   VAR
      sFB_Displacement010 { ExternalAccessible := 'False'; ExternalVisible := 'False'; ExternalWritable := 'False'; S7_SetPoint := 'False'} : "FB_Displacement";   // Displacement calculation for 010 conveyor
      sFB_Displacement020 { ExternalAccessible := 'False'; ExternalVisible := 'False'; ExternalWritable := 'False'; S7_SetPoint := 'False'} : "FB_Displacement";   // Displacement calculation for 020 conveyor
      sFB_Displacement030 { ExternalAccessible := 'False'; ExternalVisible := 'False'; ExternalWritable := 'False'; S7_SetPoint := 'False'} : "FB_Displacement";   // Displacement calculation for 030 conveyor
      sFB_Displacement040 { ExternalAccessible := 'False'; ExternalVisible := 'False'; ExternalWritable := 'False'; S7_SetPoint := 'False'} : "FB_Displacement";   // Displacement calculation for 040 conveyor
      sFB_Displacement050 { ExternalAccessible := 'False'; ExternalVisible := 'False'; ExternalWritable := 'False'; S7_SetPoint := 'False'} : "FB_Displacement";   // Displacement calculation for 050 conveyor
      sFB_Displacement060 { ExternalAccessible := 'False'; ExternalVisible := 'False'; ExternalWritable := 'False'; S7_SetPoint := 'False'} : "FB_Displacement";   // Displacement calculation for 060 conveyor
      sFB_Displacement070 { ExternalAccessible := 'False'; ExternalVisible := 'False'; ExternalWritable := 'False'; S7_SetPoint := 'False'} : "FB_Displacement";   // Displacement calculation for 070 conveyor
      sFB_Displacement080 { ExternalAccessible := 'False'; ExternalVisible := 'False'; ExternalWritable := 'False'; S7_SetPoint := 'False'} : "FB_Displacement";   // Displacement calculation for 080 conveyor
      sFB_Displacement090 { ExternalAccessible := 'False'; ExternalVisible := 'False'; ExternalWritable := 'False'; S7_SetPoint := 'False'} : "FB_Displacement";   // Displacement calculation for 090 conveyor
      sFB_Displacement100 { ExternalAccessible := 'False'; ExternalVisible := 'False'; ExternalWritable := 'False'; S7_SetPoint := 'False'} : "FB_Displacement";   // Displacement calculation for 100 conveyor
      sFB_Displacement110 { ExternalAccessible := 'False'; ExternalVisible := 'False'; ExternalWritable := 'False'; S7_SetPoint := 'False'} : "FB_Displacement";   // Displacement calculation for 110 conveyor
      sFB_Displacement120 { ExternalAccessible := 'False'; ExternalVisible := 'False'; ExternalWritable := 'False'; S7_SetPoint := 'False'} : "FB_Displacement";   // Displacement calculation for 120 conveyor
      sFB_Displacement121 { ExternalAccessible := 'False'; ExternalVisible := 'False'; ExternalWritable := 'False'; S7_SetPoint := 'False'} : "FB_Displacement";   // Displacement calculation for 121 conveyor
      sFB_Displacement210 { ExternalAccessible := 'False'; ExternalVisible := 'False'; ExternalWritable := 'False'; S7_SetPoint := 'False'} : "FB_Displacement";   // Displacement calculation for 210 conveyor
      sFB_Displacement220 { ExternalAccessible := 'False'; ExternalVisible := 'False'; ExternalWritable := 'False'; S7_SetPoint := 'False'} : "FB_Displacement";   // Displacement calculation for 220 conveyor
      sFB_Displacement221 { ExternalAccessible := 'False'; ExternalVisible := 'False'; ExternalWritable := 'False'; S7_SetPoint := 'False'} : "FB_Displacement";   // Displacement calculation for 221 conveyor
      sFB_Displacement230 { ExternalAccessible := 'False'; ExternalVisible := 'False'; ExternalWritable := 'False'; S7_SetPoint := 'False'} : "FB_Displacement";   // Displacement calculation for 230 conveyor
      sFB_Displacement240 { ExternalAccessible := 'False'; ExternalVisible := 'False'; ExternalWritable := 'False'; S7_SetPoint := 'False'} : "FB_Displacement";   // Displacement calculation for 240 conveyor
      sFB_Displacement250 { ExternalAccessible := 'False'; ExternalVisible := 'False'; ExternalWritable := 'False'; S7_SetPoint := 'False'} : "FB_Displacement";   // Displacement calculation for 250 conveyor
      sFB_Displacement260 { ExternalAccessible := 'False'; ExternalVisible := 'False'; ExternalWritable := 'False'; S7_SetPoint := 'False'} : "FB_Displacement";   // Displacement calculation for 260 conveyor
      sFB_Displacement270 { ExternalAccessible := 'False'; ExternalVisible := 'False'; ExternalWritable := 'False'; S7_SetPoint := 'False'} : "FB_Displacement";   // Displacement calculation for 270 conveyor
      sFB_Displacement280 { ExternalAccessible := 'False'; ExternalVisible := 'False'; ExternalWritable := 'False'; S7_SetPoint := 'False'} : "FB_Displacement";   // Displacement calculation for 280 conveyor
      sFB_Displacement290 { ExternalAccessible := 'False'; ExternalVisible := 'False'; ExternalWritable := 'False'; S7_SetPoint := 'False'} : "FB_Displacement";   // Displacement calculation for 290 conveyor
      sFB_Displacement291 { ExternalAccessible := 'False'; ExternalVisible := 'False'; ExternalWritable := 'False'; S7_SetPoint := 'False'} : "FB_Displacement";   // Displacement calculation for 291 conveyor
      sFB_Displacement300 { ExternalAccessible := 'False'; ExternalVisible := 'False'; ExternalWritable := 'False'; S7_SetPoint := 'False'} : "FB_Displacement";   // Displacement calculation for 300 conveyor
      sFB_Displacement410 { ExternalAccessible := 'False'; ExternalVisible := 'False'; ExternalWritable := 'False'; S7_SetPoint := 'False'} : "FB_Displacement";   // Displacement calculation for 410 conveyor
      sFB_Displacement420 { ExternalAccessible := 'False'; ExternalVisible := 'False'; ExternalWritable := 'False'; S7_SetPoint := 'False'} : "FB_Displacement";   // Displacement calculation for 420 conveyor
      sFB_Displacement421 { ExternalAccessible := 'False'; ExternalVisible := 'False'; ExternalWritable := 'False'; S7_SetPoint := 'False'} : "FB_Displacement";   // Displacement calculation for 421 conveyor
      sFB_Displacement430 { ExternalAccessible := 'False'; ExternalVisible := 'False'; ExternalWritable := 'False'; S7_SetPoint := 'False'} : "FB_Displacement";   // Displacement calculation for 430 conveyor
      sFB_Displacement440 { ExternalAccessible := 'False'; ExternalVisible := 'False'; ExternalWritable := 'False'; S7_SetPoint := 'False'} : "FB_Displacement";   // Displacement calculation for 440 conveyor
      sFB_Displacement450 { ExternalAccessible := 'False'; ExternalVisible := 'False'; ExternalWritable := 'False'; S7_SetPoint := 'False'} : "FB_Displacement";   // Displacement calculation for 450 conveyor
      sFB_Displacement460 { ExternalAccessible := 'False'; ExternalVisible := 'False'; ExternalWritable := 'False'; S7_SetPoint := 'False'} : "FB_Displacement";   // Displacement calculation for 460 conveyor
      sFB_Displacement470 { ExternalAccessible := 'False'; ExternalVisible := 'False'; ExternalWritable := 'False'; S7_SetPoint := 'False'} : "FB_Displacement";   // Displacement calculation for 470 conveyor
      sFB_Displacement480 { ExternalAccessible := 'False'; ExternalVisible := 'False'; ExternalWritable := 'False'; S7_SetPoint := 'False'} : "FB_Displacement";   // Displacement calculation for 480 conveyor
      sFB_Displacement490 { ExternalAccessible := 'False'; ExternalVisible := 'False'; ExternalWritable := 'False'; S7_SetPoint := 'False'} : "FB_Displacement";   // Displacement calculation for 490 conveyor
      sFB_Displacement491 { ExternalAccessible := 'False'; ExternalVisible := 'False'; ExternalWritable := 'False'; S7_SetPoint := 'False'} : "FB_Displacement";   // Displacement calculation for 491 conveyor
      sFB_Displacement500 { ExternalAccessible := 'False'; ExternalVisible := 'False'; ExternalWritable := 'False'; S7_SetPoint := 'False'} : "FB_Displacement";   // Displacement calculation for 500 conveyor
      sFB_Displacement610 { ExternalAccessible := 'False'; ExternalVisible := 'False'; ExternalWritable := 'False'; S7_SetPoint := 'False'} : "FB_Displacement";   // Displacement calculation for 610 conveyor
      sFB_Displacement611 { ExternalAccessible := 'False'; ExternalVisible := 'False'; ExternalWritable := 'False'; S7_SetPoint := 'False'} : "FB_Displacement";   // Displacement calculation for 611 conveyor
      sFB_Displacement620 { ExternalAccessible := 'False'; ExternalVisible := 'False'; ExternalWritable := 'False'; S7_SetPoint := 'False'} : "FB_Displacement";   // Displacement calculation for 620 conveyor
      sFB_Displacement630 { ExternalAccessible := 'False'; ExternalVisible := 'False'; ExternalWritable := 'False'; S7_SetPoint := 'False'} : "FB_Displacement";   // Displacement calculation for 630 conveyor
      sFB_Displacement640 { ExternalAccessible := 'False'; ExternalVisible := 'False'; ExternalWritable := 'False'; S7_SetPoint := 'False'} : "FB_Displacement";   // Displacement calculation for 640 conveyor
      sUDT_Interface010 { ExternalAccessible := 'False'; ExternalVisible := 'False'; ExternalWritable := 'False'; S7_SetPoint := 'False'} : "UDT_ConveyorInterface";   // Interface structure for 010 conveyor
      sUDT_Interface020 { ExternalAccessible := 'False'; ExternalVisible := 'False'; ExternalWritable := 'False'; S7_SetPoint := 'False'} : "UDT_ConveyorInterface";   // Interface structure for 020 conveyor
      sUDT_Interface030 { ExternalAccessible := 'False'; ExternalVisible := 'False'; ExternalWritable := 'False'; S7_SetPoint := 'False'} : "UDT_ConveyorInterface";   // Interface structure for 030 conveyor
      sUDT_Interface040 { ExternalAccessible := 'False'; ExternalVisible := 'False'; ExternalWritable := 'False'; S7_SetPoint := 'False'} : "UDT_ConveyorInterface";   // Interface structure for 040 conveyor
      sUDT_Interface050 { ExternalAccessible := 'False'; ExternalVisible := 'False'; ExternalWritable := 'False'; S7_SetPoint := 'False'} : "UDT_ConveyorInterface";   // Interface structure for 050 conveyor
      sUDT_Interface060 { ExternalAccessible := 'False'; ExternalVisible := 'False'; ExternalWritable := 'False'; S7_SetPoint := 'False'} : "UDT_ConveyorInterface";   // Interface structure for 060 conveyor
      sUDT_Interface070 { ExternalAccessible := 'False'; ExternalVisible := 'False'; ExternalWritable := 'False'; S7_SetPoint := 'False'} : "UDT_ConveyorInterface";   // Interface structure for 070 conveyor
      sUDT_Interface080 { ExternalAccessible := 'False'; ExternalVisible := 'False'; ExternalWritable := 'False'; S7_SetPoint := 'False'} : "UDT_ConveyorInterface";   // Interface structure for 080 conveyor
      sUDT_Interface090 { ExternalAccessible := 'False'; ExternalVisible := 'False'; ExternalWritable := 'False'; S7_SetPoint := 'False'} : "UDT_ConveyorInterface";   // Interface structure for 090 conveyor
      sUDT_Interface100 { ExternalAccessible := 'False'; ExternalVisible := 'False'; ExternalWritable := 'False'; S7_SetPoint := 'False'} : "UDT_ConveyorInterface";   // Interface structure for 100 conveyor
      sUDT_Interface110 { ExternalAccessible := 'False'; ExternalVisible := 'False'; ExternalWritable := 'False'; S7_SetPoint := 'False'} : "UDT_ConveyorInterface";   // Interface structure for 110 conveyor
      sUDT_Interface120 { ExternalAccessible := 'False'; ExternalVisible := 'False'; ExternalWritable := 'False'; S7_SetPoint := 'False'} : "UDT_ConveyorInterface";   // Interface structure for 120 conveyor
      sUDT_Interface121 { ExternalAccessible := 'False'; ExternalVisible := 'False'; ExternalWritable := 'False'; S7_SetPoint := 'False'} : "UDT_ConveyorInterface";   // Interface structure for 121 conveyor
      sUDT_Interface210 { ExternalAccessible := 'False'; ExternalVisible := 'False'; ExternalWritable := 'False'; S7_SetPoint := 'False'} : "UDT_ConveyorInterface";   // Interface structure for 210 conveyor
      sUDT_Interface220 { ExternalAccessible := 'False'; ExternalVisible := 'False'; ExternalWritable := 'False'; S7_SetPoint := 'False'} : "UDT_ConveyorInterface";   // Interface structure for 220 conveyor
      sUDT_Interface221 { ExternalAccessible := 'False'; ExternalVisible := 'False'; ExternalWritable := 'False'; S7_SetPoint := 'False'} : "UDT_ConveyorInterface";   // Interface structure for 221 conveyor
      sUDT_Interface230 { ExternalAccessible := 'False'; ExternalVisible := 'False'; ExternalWritable := 'False'; S7_SetPoint := 'False'} : "UDT_ConveyorInterface";   // Interface structure for 230 conveyor
      sUDT_Interface240 { ExternalAccessible := 'False'; ExternalVisible := 'False'; ExternalWritable := 'False'; S7_SetPoint := 'False'} : "UDT_ConveyorInterface";   // Interface structure for 240 conveyor
      sUDT_Interface250 { ExternalAccessible := 'False'; ExternalVisible := 'False'; ExternalWritable := 'False'; S7_SetPoint := 'False'} : "UDT_ConveyorInterface";   // Interface structure for 250 conveyor
      sUDT_Interface260 { ExternalAccessible := 'False'; ExternalVisible := 'False'; ExternalWritable := 'False'; S7_SetPoint := 'False'} : "UDT_ConveyorInterface";   // Interface structure for 260 conveyor
      sUDT_Interface270 { ExternalAccessible := 'False'; ExternalVisible := 'False'; ExternalWritable := 'False'; S7_SetPoint := 'False'} : "UDT_ConveyorInterface";   // Interface structure for 270 conveyor
      sUDT_Interface280 { ExternalAccessible := 'False'; ExternalVisible := 'False'; ExternalWritable := 'False'; S7_SetPoint := 'False'} : "UDT_ConveyorInterface";   // Interface structure for 280 conveyor
      sUDT_Interface290 { ExternalAccessible := 'False'; ExternalVisible := 'False'; ExternalWritable := 'False'; S7_SetPoint := 'False'} : "UDT_ConveyorInterface";   // Interface structure for 290 conveyor
      sUDT_Interface291 { ExternalAccessible := 'False'; ExternalVisible := 'False'; ExternalWritable := 'False'; S7_SetPoint := 'False'} : "UDT_ConveyorInterface";   // Interface structure for 291 conveyor
      sUDT_Interface300 { ExternalAccessible := 'False'; ExternalVisible := 'False'; ExternalWritable := 'False'; S7_SetPoint := 'False'} : "UDT_ConveyorInterface";   // Interface structure for 300 conveyor
      sUDT_Interface410 { ExternalAccessible := 'False'; ExternalVisible := 'False'; ExternalWritable := 'False'; S7_SetPoint := 'False'} : "UDT_ConveyorInterface";   // Interface structure for 410 conveyor
      sUDT_Interface420 { ExternalAccessible := 'False'; ExternalVisible := 'False'; ExternalWritable := 'False'; S7_SetPoint := 'False'} : "UDT_ConveyorInterface";   // Interface structure for 420 conveyor
      sUDT_Interface421 { ExternalAccessible := 'False'; ExternalVisible := 'False'; ExternalWritable := 'False'; S7_SetPoint := 'False'} : "UDT_ConveyorInterface";   // Interface structure for 421 conveyor
      sUDT_Interface430 { ExternalAccessible := 'False'; ExternalVisible := 'False'; ExternalWritable := 'False'; S7_SetPoint := 'False'} : "UDT_ConveyorInterface";   // Interface structure for 430 conveyor
      sUDT_Interface440 { ExternalAccessible := 'False'; ExternalVisible := 'False'; ExternalWritable := 'False'; S7_SetPoint := 'False'} : "UDT_ConveyorInterface";   // Interface structure for 440 conveyor
      sUDT_Interface450 { ExternalAccessible := 'False'; ExternalVisible := 'False'; ExternalWritable := 'False'; S7_SetPoint := 'False'} : "UDT_ConveyorInterface";   // Interface structure for 450 conveyor
      sUDT_Interface460 { ExternalAccessible := 'False'; ExternalVisible := 'False'; ExternalWritable := 'False'; S7_SetPoint := 'False'} : "UDT_ConveyorInterface";   // Interface structure for 460 conveyor
      sUDT_Interface470 { ExternalAccessible := 'False'; ExternalVisible := 'False'; ExternalWritable := 'False'; S7_SetPoint := 'False'} : "UDT_ConveyorInterface";   // Interface structure for 470 conveyor
      sUDT_Interface480 { ExternalAccessible := 'False'; ExternalVisible := 'False'; ExternalWritable := 'False'; S7_SetPoint := 'False'} : "UDT_ConveyorInterface";   // Interface structure for 480 conveyor
      sUDT_Interface490 { ExternalAccessible := 'False'; ExternalVisible := 'False'; ExternalWritable := 'False'; S7_SetPoint := 'False'} : "UDT_ConveyorInterface";   // Interface structure for 490 conveyor
      sUDT_Interface491 { ExternalAccessible := 'False'; ExternalVisible := 'False'; ExternalWritable := 'False'; S7_SetPoint := 'False'} : "UDT_ConveyorInterface";   // Interface structure for 491 conveyor
      sUDT_Interface500 { ExternalAccessible := 'False'; ExternalVisible := 'False'; ExternalWritable := 'False'; S7_SetPoint := 'False'} : "UDT_ConveyorInterface";   // Interface structure for 500 conveyor
      sUDT_Interface610 { ExternalAccessible := 'False'; ExternalVisible := 'False'; ExternalWritable := 'False'; S7_SetPoint := 'False'} : "UDT_ConveyorInterface";   // Interface structure for 610 conveyor
      sUDT_Interface611 { ExternalAccessible := 'False'; ExternalVisible := 'False'; ExternalWritable := 'False'; S7_SetPoint := 'False'} : "UDT_ConveyorInterface";   // Interface structure for 611 conveyor
      sUDT_Interface620 { ExternalAccessible := 'False'; ExternalVisible := 'False'; ExternalWritable := 'False'; S7_SetPoint := 'False'} : "UDT_ConveyorInterface";   // Interface structure for 620 conveyor
      sUDT_Interface630 { ExternalAccessible := 'False'; ExternalVisible := 'False'; ExternalWritable := 'False'; S7_SetPoint := 'False'} : "UDT_ConveyorInterface";   // Interface structure for 630 conveyor
      sUDT_Interface640 { ExternalAccessible := 'False'; ExternalVisible := 'False'; ExternalWritable := 'False'; S7_SetPoint := 'False'} : "UDT_ConveyorInterface";   // Interface structure for 640 conveyor
      sUDT_Handshake010 { ExternalAccessible := 'False'; ExternalVisible := 'False'; ExternalWritable := 'False'; S7_SetPoint := 'False'} : "UDT_ConveyorHandshake";   // Handshake structure for 010 conveyor
      sUDT_Handshake020 { ExternalAccessible := 'False'; ExternalVisible := 'False'; ExternalWritable := 'False'; S7_SetPoint := 'False'} : "UDT_ConveyorHandshake";   // Handshake structure for 020 conveyor
      sUDT_Handshake030 { ExternalAccessible := 'False'; ExternalVisible := 'False'; ExternalWritable := 'False'; S7_SetPoint := 'False'} : "UDT_ConveyorHandshake";   // Handshake structure for 030 conveyor
      sUDT_Handshake040 { ExternalAccessible := 'False'; ExternalVisible := 'False'; ExternalWritable := 'False'; S7_SetPoint := 'False'} : "UDT_ConveyorHandshake";   // Handshake structure for 040 conveyor
      sUDT_Handshake050 { ExternalAccessible := 'False'; ExternalVisible := 'False'; ExternalWritable := 'False'; S7_SetPoint := 'False'} : "UDT_ConveyorHandshake";   // Handshake structure for 050 conveyor
      sUDT_Handshake060 { ExternalAccessible := 'False'; ExternalVisible := 'False'; ExternalWritable := 'False'; S7_SetPoint := 'False'} : "UDT_ConveyorHandshake";   // Handshake structure for 060 conveyor
      sUDT_Handshake070 { ExternalAccessible := 'False'; ExternalVisible := 'False'; ExternalWritable := 'False'; S7_SetPoint := 'False'} : "UDT_ConveyorHandshake";   // Handshake structure for 070 conveyor
      sUDT_Handshake080 { ExternalAccessible := 'False'; ExternalVisible := 'False'; ExternalWritable := 'False'; S7_SetPoint := 'False'} : "UDT_ConveyorHandshake";   // Handshake structure for 080 conveyor
      sUDT_Handshake090 { ExternalAccessible := 'False'; ExternalVisible := 'False'; ExternalWritable := 'False'; S7_SetPoint := 'False'} : "UDT_ConveyorHandshake";   // Handshake structure for 090 conveyor
      sUDT_Handshake100 { ExternalAccessible := 'False'; ExternalVisible := 'False'; ExternalWritable := 'False'; S7_SetPoint := 'False'} : "UDT_ConveyorHandshake";   // Handshake structure for 100 conveyor
      sUDT_Handshake110 { ExternalAccessible := 'False'; ExternalVisible := 'False'; ExternalWritable := 'False'; S7_SetPoint := 'False'} : "UDT_ConveyorHandshake";   // Handshake structure for 110 conveyor
      sUDT_Handshake120 { ExternalAccessible := 'False'; ExternalVisible := 'False'; ExternalWritable := 'False'; S7_SetPoint := 'False'} : "UDT_ConveyorHandshake";   // Handshake structure for 120 conveyor
      sUDT_Handshake121 { ExternalAccessible := 'False'; ExternalVisible := 'False'; ExternalWritable := 'False'; S7_SetPoint := 'False'} : "UDT_ConveyorHandshake";   // Handshake structure for 121 conveyor
      sUDT_HandshakeUp121 { ExternalAccessible := 'False'; ExternalVisible := 'False'; ExternalWritable := 'False'; S7_SetPoint := 'False'} : "UDT_ConveyorHandshake";   // HandshakeUp structure for 121 conveyor
      sUDT_Handshake210 { ExternalAccessible := 'False'; ExternalVisible := 'False'; ExternalWritable := 'False'; S7_SetPoint := 'False'} : "UDT_ConveyorHandshake";   // Handshake structure for 210 conveyor
      sUDT_Handshake220 { ExternalAccessible := 'False'; ExternalVisible := 'False'; ExternalWritable := 'False'; S7_SetPoint := 'False'} : "UDT_ConveyorHandshake";   // Handshake structure for 220 conveyor
      sUDT_Handshake221 { ExternalAccessible := 'False'; ExternalVisible := 'False'; ExternalWritable := 'False'; S7_SetPoint := 'False'} : "UDT_ConveyorHandshake";   // Handshake structure for 221 conveyor
      sUDT_Handshake230 { ExternalAccessible := 'False'; ExternalVisible := 'False'; ExternalWritable := 'False'; S7_SetPoint := 'False'} : "UDT_ConveyorHandshake";   // Handshake structure for 230 conveyor
      sUDT_Handshake240 { ExternalAccessible := 'False'; ExternalVisible := 'False'; ExternalWritable := 'False'; S7_SetPoint := 'False'} : "UDT_ConveyorHandshake";   // Handshake structure for 240 conveyor
      sUDT_Handshake250 { ExternalAccessible := 'False'; ExternalVisible := 'False'; ExternalWritable := 'False'; S7_SetPoint := 'False'} : "UDT_ConveyorHandshake";   // Handshake structure for 250 conveyor
      sUDT_Handshake260 { ExternalAccessible := 'False'; ExternalVisible := 'False'; ExternalWritable := 'False'; S7_SetPoint := 'False'} : "UDT_ConveyorHandshake";   // Handshake structure for 260 conveyor
      sUDT_Handshake270 { ExternalAccessible := 'False'; ExternalVisible := 'False'; ExternalWritable := 'False'; S7_SetPoint := 'False'} : "UDT_ConveyorHandshake";   // Handshake structure for 270 conveyor
      sUDT_Handshake280 { ExternalAccessible := 'False'; ExternalVisible := 'False'; ExternalWritable := 'False'; S7_SetPoint := 'False'} : "UDT_ConveyorHandshake";   // Handshake structure for 280 conveyor
      sUDT_Handshake290 { ExternalAccessible := 'False'; ExternalVisible := 'False'; ExternalWritable := 'False'; S7_SetPoint := 'False'} : "UDT_ConveyorHandshake";   // Handshake structure for 290 conveyor
      sUDT_Handshake291 { ExternalAccessible := 'False'; ExternalVisible := 'False'; ExternalWritable := 'False'; S7_SetPoint := 'False'} : "UDT_ConveyorHandshake";   // Handshake structure for 291 conveyor
      sUDT_HandshakeUp291 { ExternalAccessible := 'False'; ExternalVisible := 'False'; ExternalWritable := 'False'; S7_SetPoint := 'False'} : "UDT_ConveyorHandshake";   // HandshakeUp structure for 291 conveyor
      sUDT_Handshake300 { ExternalAccessible := 'False'; ExternalVisible := 'False'; ExternalWritable := 'False'; S7_SetPoint := 'False'} : "UDT_ConveyorHandshake";   // Handshake structure for 300 conveyor
      sUDT_Handshake410 { ExternalAccessible := 'False'; ExternalVisible := 'False'; ExternalWritable := 'False'; S7_SetPoint := 'False'} : "UDT_ConveyorHandshake";   // Handshake structure for 410 conveyor
      sUDT_Handshake420 { ExternalAccessible := 'False'; ExternalVisible := 'False'; ExternalWritable := 'False'; S7_SetPoint := 'False'} : "UDT_ConveyorHandshake";   // Handshake structure for 420 conveyor
      sUDT_Handshake421 { ExternalAccessible := 'False'; ExternalVisible := 'False'; ExternalWritable := 'False'; S7_SetPoint := 'False'} : "UDT_ConveyorHandshake";   // Handshake structure for 421 conveyor
      sUDT_Handshake430 { ExternalAccessible := 'False'; ExternalVisible := 'False'; ExternalWritable := 'False'; S7_SetPoint := 'False'} : "UDT_ConveyorHandshake";   // Handshake structure for 430 conveyor
      sUDT_Handshake440 { ExternalAccessible := 'False'; ExternalVisible := 'False'; ExternalWritable := 'False'; S7_SetPoint := 'False'} : "UDT_ConveyorHandshake";   // Handshake structure for 440 conveyor
      sUDT_Handshake450 { ExternalAccessible := 'False'; ExternalVisible := 'False'; ExternalWritable := 'False'; S7_SetPoint := 'False'} : "UDT_ConveyorHandshake";   // Handshake structure for 450 conveyor
      sUDT_Handshake460 { ExternalAccessible := 'False'; ExternalVisible := 'False'; ExternalWritable := 'False'; S7_SetPoint := 'False'} : "UDT_ConveyorHandshake";   // Handshake structure for 460 conveyor
      sUDT_Handshake470 { ExternalAccessible := 'False'; ExternalVisible := 'False'; ExternalWritable := 'False'; S7_SetPoint := 'False'} : "UDT_ConveyorHandshake";   // Handshake structure for 470 conveyor
      sUDT_Handshake480 { ExternalAccessible := 'False'; ExternalVisible := 'False'; ExternalWritable := 'False'; S7_SetPoint := 'False'} : "UDT_ConveyorHandshake";   // Handshake structure for 480 conveyor
      sUDT_Handshake490 { ExternalAccessible := 'False'; ExternalVisible := 'False'; ExternalWritable := 'False'; S7_SetPoint := 'False'} : "UDT_ConveyorHandshake";   // Handshake structure for 490 conveyor
      sUDT_Handshake491 { ExternalAccessible := 'False'; ExternalVisible := 'False'; ExternalWritable := 'False'; S7_SetPoint := 'False'} : "UDT_ConveyorHandshake";   // Handshake structure for 491 conveyor
      sUDT_Handshake500 { ExternalAccessible := 'False'; ExternalVisible := 'False'; ExternalWritable := 'False'; S7_SetPoint := 'False'} : "UDT_ConveyorHandshake";   // Handshake structure for 500 conveyor
      sUDT_Handshake610 { ExternalAccessible := 'False'; ExternalVisible := 'False'; ExternalWritable := 'False'; S7_SetPoint := 'False'} : "UDT_ConveyorHandshake";   // Handshake structure for 610 conveyor
      sUDT_Handshake611 { ExternalAccessible := 'False'; ExternalVisible := 'False'; ExternalWritable := 'False'; S7_SetPoint := 'False'} : "UDT_ConveyorHandshake";   // Handshake structure for 611 conveyor
      sUDT_Handshake620 { ExternalAccessible := 'False'; ExternalVisible := 'False'; ExternalWritable := 'False'; S7_SetPoint := 'False'} : "UDT_ConveyorHandshake";   // Handshake structure for 620 conveyor
      sUDT_Handshake630 { ExternalAccessible := 'False'; ExternalVisible := 'False'; ExternalWritable := 'False'; S7_SetPoint := 'False'} : "UDT_ConveyorHandshake";   // Handshake structure for 630 conveyor
      sUDT_Handshake640 { ExternalAccessible := 'False'; ExternalVisible := 'False'; ExternalWritable := 'False'; S7_SetPoint := 'False'} : "UDT_ConveyorHandshake";   // Handshake structure for 640 conveyor
      sFB_PEC010 { ExternalAccessible := 'False'; ExternalVisible := 'False'; ExternalWritable := 'False'; S7_SetPoint := 'False'} : "FB_PEC";   // Photoeye handling for 010 conveyor
      sFB_PEC020 { ExternalAccessible := 'False'; ExternalVisible := 'False'; ExternalWritable := 'False'; S7_SetPoint := 'False'} : "FB_PEC";   // Photoeye handling for 020 conveyor
      sFB_PEC040 { ExternalAccessible := 'False'; ExternalVisible := 'False'; ExternalWritable := 'False'; S7_SetPoint := 'False'} : "FB_PEC";   // Photoeye handling for 040 conveyor
      sFB_PEC050 { ExternalAccessible := 'False'; ExternalVisible := 'False'; ExternalWritable := 'False'; S7_SetPoint := 'False'} : "FB_PEC";   // Photoeye handling for 050 conveyor
      sFB_PEC060 { ExternalAccessible := 'False'; ExternalVisible := 'False'; ExternalWritable := 'False'; S7_SetPoint := 'False'} : "FB_PEC";   // Photoeye handling for 060 conveyor
      sFB_PEC070 { ExternalAccessible := 'False'; ExternalVisible := 'False'; ExternalWritable := 'False'; S7_SetPoint := 'False'} : "FB_PEC";   // Photoeye handling for 070 conveyor
      sFB_PEC080 { ExternalAccessible := 'False'; ExternalVisible := 'False'; ExternalWritable := 'False'; S7_SetPoint := 'False'} : "FB_PEC";   // Photoeye handling for 080 conveyor
      sFB_PEC100 { ExternalAccessible := 'False'; ExternalVisible := 'False'; ExternalWritable := 'False'; S7_SetPoint := 'False'} : "FB_PEC";   // Photoeye handling for 100 conveyor
      sFB_PEC110 { ExternalAccessible := 'False'; ExternalVisible := 'False'; ExternalWritable := 'False'; S7_SetPoint := 'False'} : "FB_PEC";   // Photoeye handling for 110 conveyor
      sFB_PEC120 { ExternalAccessible := 'False'; ExternalVisible := 'False'; ExternalWritable := 'False'; S7_SetPoint := 'False'} : "FB_PEC";   // Photoeye handling for 120 conveyor
      sFB_PEC210 { ExternalAccessible := 'False'; ExternalVisible := 'False'; ExternalWritable := 'False'; S7_SetPoint := 'False'} : "FB_PEC";   // Photoeye handling for 210 conveyor
      sFB_PEC220 { ExternalAccessible := 'False'; ExternalVisible := 'False'; ExternalWritable := 'False'; S7_SetPoint := 'False'} : "FB_PEC";   // Photoeye handling for 220 conveyor
      sFB_PEC240 { ExternalAccessible := 'False'; ExternalVisible := 'False'; ExternalWritable := 'False'; S7_SetPoint := 'False'} : "FB_PEC";   // Photoeye handling for 240 conveyor
      sFB_PEC250 { ExternalAccessible := 'False'; ExternalVisible := 'False'; ExternalWritable := 'False'; S7_SetPoint := 'False'} : "FB_PEC";   // Photoeye handling for 250 conveyor
      sFB_PEC260 { ExternalAccessible := 'False'; ExternalVisible := 'False'; ExternalWritable := 'False'; S7_SetPoint := 'False'} : "FB_PEC";   // Photoeye handling for 260 conveyor
      sFB_PEC280 { ExternalAccessible := 'False'; ExternalVisible := 'False'; ExternalWritable := 'False'; S7_SetPoint := 'False'} : "FB_PEC";   // Photoeye handling for 280 conveyor
      sFB_PEC290 { ExternalAccessible := 'False'; ExternalVisible := 'False'; ExternalWritable := 'False'; S7_SetPoint := 'False'} : "FB_PEC";   // Photoeye handling for 290 conveyor
      sFB_PEC300 { ExternalAccessible := 'False'; ExternalVisible := 'False'; ExternalWritable := 'False'; S7_SetPoint := 'False'} : "FB_PEC";   // Photoeye handling for 3000 conveyor
      sFB_PEC410 { ExternalAccessible := 'False'; ExternalVisible := 'False'; ExternalWritable := 'False'; S7_SetPoint := 'False'} : "FB_PEC";   // Photoeye handling for 410 conveyor
      sFB_PEC420 { ExternalAccessible := 'False'; ExternalVisible := 'False'; ExternalWritable := 'False'; S7_SetPoint := 'False'} : "FB_PEC";   // Photoeye handling for 420 conveyor
      sFB_PEC440 { ExternalAccessible := 'False'; ExternalVisible := 'False'; ExternalWritable := 'False'; S7_SetPoint := 'False'} : "FB_PEC";   // Photoeye handling for 440 conveyor
      sFB_PEC450 { ExternalAccessible := 'False'; ExternalVisible := 'False'; ExternalWritable := 'False'; S7_SetPoint := 'False'} : "FB_PEC";   // Photoeye handling for 450 conveyor
      sFB_PEC460 { ExternalAccessible := 'False'; ExternalVisible := 'False'; ExternalWritable := 'False'; S7_SetPoint := 'False'} : "FB_PEC";   // Photoeye handling for 460 conveyor
      sFB_PEC480 { ExternalAccessible := 'False'; ExternalVisible := 'False'; ExternalWritable := 'False'; S7_SetPoint := 'False'} : "FB_PEC";   // Photoeye handling for 480 conveyor
      sFB_PEC490 { ExternalAccessible := 'False'; ExternalVisible := 'False'; ExternalWritable := 'False'; S7_SetPoint := 'False'} : "FB_PEC";   // Photoeye handling for 490 conveyor
      sFB_PEC500 { ExternalAccessible := 'False'; ExternalVisible := 'False'; ExternalWritable := 'False'; S7_SetPoint := 'False'} : "FB_PEC";   // Photoeye handling for 500 conveyor
      sFB_PEC610 { ExternalAccessible := 'False'; ExternalVisible := 'False'; ExternalWritable := 'False'; S7_SetPoint := 'False'} : "FB_PEC";   // Photoeye handling for 610 conveyor
      sFB_PEC640 { ExternalAccessible := 'False'; ExternalVisible := 'False'; ExternalWritable := 'False'; S7_SetPoint := 'False'} : "FB_PEC";   // Photoeye handling for 640 conveyor
      sFB_Conveyor010 { ExternalAccessible := 'False'; ExternalVisible := 'False'; ExternalWritable := 'False'; S7_SetPoint := 'False'} : "FB_Conveyor";   // Function block to control the 010 conveyor
      sFB_Conveyor020 { ExternalAccessible := 'False'; ExternalVisible := 'False'; ExternalWritable := 'False'; S7_SetPoint := 'False'} : "FB_Conveyor";   // Function block to control the 020 conveyor
      sFB_Conveyor030 { ExternalAccessible := 'False'; ExternalVisible := 'False'; ExternalWritable := 'False'; S7_SetPoint := 'False'} : "FB_Conveyor";   // Function block to control the 030 conveyor
      sFB_Conveyor040 { ExternalAccessible := 'False'; ExternalVisible := 'False'; ExternalWritable := 'False'; S7_SetPoint := 'False'} : "FB_Conveyor";   // Function block to control the 040 conveyor
      sFB_Conveyor050 { ExternalAccessible := 'False'; ExternalVisible := 'False'; ExternalWritable := 'False'; S7_SetPoint := 'False'} : "FB_Conveyor";   // Function block to control the 050 conveyor
      sFB_Conveyor060 { ExternalAccessible := 'False'; ExternalVisible := 'False'; ExternalWritable := 'False'; S7_SetPoint := 'False'} : "FB_Conveyor";   // Function block to control the 060 conveyor
      sFB_Conveyor070 { ExternalAccessible := 'False'; ExternalVisible := 'False'; ExternalWritable := 'False'; S7_SetPoint := 'False'} : "FB_Conveyor";   // Function block to control the 070 conveyor
      sFB_Conveyor080 { ExternalAccessible := 'False'; ExternalVisible := 'False'; ExternalWritable := 'False'; S7_SetPoint := 'False'} : "FB_Conveyor";   // Function block to control the 080 conveyor
      sFB_Conveyor090 { ExternalAccessible := 'False'; ExternalVisible := 'False'; ExternalWritable := 'False'; S7_SetPoint := 'False'} : "FB_Conveyor";   // Function block to control the 090 conveyor
      sFB_Conveyor100 { ExternalAccessible := 'False'; ExternalVisible := 'False'; ExternalWritable := 'False'; S7_SetPoint := 'False'} : "FB_Conveyor";   // Function block to control the 100 conveyor
      sFB_Conveyor110 { ExternalAccessible := 'False'; ExternalVisible := 'False'; ExternalWritable := 'False'; S7_SetPoint := 'False'} : "FB_Conveyor";   // Function block to control the 110 conveyor
      sFB_Conveyor210 { ExternalAccessible := 'False'; ExternalVisible := 'False'; ExternalWritable := 'False'; S7_SetPoint := 'False'} : "FB_Conveyor";   // Function block to control the 210 conveyor
      sFB_Conveyor230 { ExternalAccessible := 'False'; ExternalVisible := 'False'; ExternalWritable := 'False'; S7_SetPoint := 'False'} : "FB_Conveyor";   // Function block to control the 230 conveyor
      sFB_Conveyor240 { ExternalAccessible := 'False'; ExternalVisible := 'False'; ExternalWritable := 'False'; S7_SetPoint := 'False'} : "FB_Conveyor";   // Function block to control the 240 conveyor
      sFB_Conveyor250 { ExternalAccessible := 'False'; ExternalVisible := 'False'; ExternalWritable := 'False'; S7_SetPoint := 'False'} : "FB_Conveyor";   // Function block to control the 250 conveyor
      sFB_Conveyor260 { ExternalAccessible := 'False'; ExternalVisible := 'False'; ExternalWritable := 'False'; S7_SetPoint := 'False'} : "FB_Conveyor";   // Function block to control the 260 conveyor
      sFB_Conveyor270 { ExternalAccessible := 'False'; ExternalVisible := 'False'; ExternalWritable := 'False'; S7_SetPoint := 'False'} : "FB_Conveyor";   // Function block to control the 270 conveyor
      sFB_Conveyor280 { ExternalAccessible := 'False'; ExternalVisible := 'False'; ExternalWritable := 'False'; S7_SetPoint := 'False'} : "FB_Conveyor";   // Function block to control the 280 conveyor
      sFB_Conveyor300 { ExternalAccessible := 'False'; ExternalVisible := 'False'; ExternalWritable := 'False'; S7_SetPoint := 'False'} : "FB_Conveyor";   // Function block to control the 300 conveyor
      sFB_Conveyor410 { ExternalAccessible := 'False'; ExternalVisible := 'False'; ExternalWritable := 'False'; S7_SetPoint := 'False'} : "FB_Conveyor";   // Function block to control the 410 conveyor
      sFB_Conveyor430 { ExternalAccessible := 'False'; ExternalVisible := 'False'; ExternalWritable := 'False'; S7_SetPoint := 'False'} : "FB_Conveyor";   // Function block to control the 430 conveyor
      sFB_Conveyor440 { ExternalAccessible := 'False'; ExternalVisible := 'False'; ExternalWritable := 'False'; S7_SetPoint := 'False'} : "FB_Conveyor";   // Function block to control the 440 conveyor
      sFB_Conveyor450 { ExternalAccessible := 'False'; ExternalVisible := 'False'; ExternalWritable := 'False'; S7_SetPoint := 'False'} : "FB_Conveyor";   // Function block to control the 450 conveyor
      sFB_Conveyor460 { ExternalAccessible := 'False'; ExternalVisible := 'False'; ExternalWritable := 'False'; S7_SetPoint := 'False'} : "FB_Conveyor";   // Function block to control the 460 conveyor
      sFB_Conveyor470 { ExternalAccessible := 'False'; ExternalVisible := 'False'; ExternalWritable := 'False'; S7_SetPoint := 'False'} : "FB_Conveyor";   // Function block to control the 470 conveyor
      sFB_Conveyor480 { ExternalAccessible := 'False'; ExternalVisible := 'False'; ExternalWritable := 'False'; S7_SetPoint := 'False'} : "FB_Conveyor";   // Function block to control the 480 conveyor
      sFB_Conveyor500 { ExternalAccessible := 'False'; ExternalVisible := 'False'; ExternalWritable := 'False'; S7_SetPoint := 'False'} : "FB_Conveyor";   // Function block to control the 500 conveyor
      sFB_Conveyor620 { ExternalAccessible := 'False'; ExternalVisible := 'False'; ExternalWritable := 'False'; S7_SetPoint := 'False'} : "FB_Conveyor";   // Function block to control the 620 conveyor
      sFB_Conveyor630 { ExternalAccessible := 'False'; ExternalVisible := 'False'; ExternalWritable := 'False'; S7_SetPoint := 'False'} : "FB_Conveyor";   // Function block to control the 630 conveyor
      sFB_Conveyor640 { ExternalAccessible := 'False'; ExternalVisible := 'False'; ExternalWritable := 'False'; S7_SetPoint := 'False'} : "FB_Conveyor";   // Function block to control the 640 conveyor
      sFB_MCOConveyLinxAixController010 { ExternalAccessible := 'False'; ExternalVisible := 'False'; ExternalWritable := 'False'; S7_SetPoint := 'False'} : "FB_MCOConveyLinxAixController";   // Function to interface with ConveyLinx Aix Controller for 010
      sFB_MCOConveyLinxAixController020 { ExternalAccessible := 'False'; ExternalVisible := 'False'; ExternalWritable := 'False'; S7_SetPoint := 'False'} : "FB_MCOConveyLinxAixController";   // Function to interface with ConveyLinx Aix Controller for 020
      sFB_MCOConveyLinxAixController030 { ExternalAccessible := 'False'; ExternalVisible := 'False'; ExternalWritable := 'False'; S7_SetPoint := 'False'} : "FB_MCOConveyLinxAixController";   // Function to interface with ConveyLinx Aix Controller for 030
      sFB_MCOConveyLinxAixController040 { ExternalAccessible := 'False'; ExternalVisible := 'False'; ExternalWritable := 'False'; S7_SetPoint := 'False'} : "FB_MCOConveyLinxAixController";   // Function to interface with ConveyLinx Aix Controller for 040
      sFB_MCOConveyLinxAixController050 { ExternalAccessible := 'False'; ExternalVisible := 'False'; ExternalWritable := 'False'; S7_SetPoint := 'False'} : "FB_MCOConveyLinxAixController";   // Function to interface with ConveyLinx Aix Controller for 050
      sFB_MCOConveyLinxAixController060 { ExternalAccessible := 'False'; ExternalVisible := 'False'; ExternalWritable := 'False'; S7_SetPoint := 'False'} : "FB_MCOConveyLinxAixController";   // Function to interface with ConveyLinx Aix Controller for 060
      sFB_MCOConveyLinxAixController070 { ExternalAccessible := 'False'; ExternalVisible := 'False'; ExternalWritable := 'False'; S7_SetPoint := 'False'} : "FB_MCOConveyLinxAixController";   // Function to interface with ConveyLinx Aix Controller for 070
      sFB_MCOConveyLinxAixController080 { ExternalAccessible := 'False'; ExternalVisible := 'False'; ExternalWritable := 'False'; S7_SetPoint := 'False'} : "FB_MCOConveyLinxAixController";   // Function to interface with ConveyLinx Aix Controller for 080
      sFB_MCOConveyLinxAixController090 { ExternalAccessible := 'False'; ExternalVisible := 'False'; ExternalWritable := 'False'; S7_SetPoint := 'False'} : "FB_MCOConveyLinxAixController";   // Function to interface with ConveyLinx Aix Controller for 090
      sFB_MCOConveyLinxAixController100 { ExternalAccessible := 'False'; ExternalVisible := 'False'; ExternalWritable := 'False'; S7_SetPoint := 'False'} : "FB_MCOConveyLinxAixController";   // Function to interface with ConveyLinx Aix Controller for 100
      sFB_MCOConveyLinxAixController110 { ExternalAccessible := 'False'; ExternalVisible := 'False'; ExternalWritable := 'False'; S7_SetPoint := 'False'} : "FB_MCOConveyLinxAixController";   // Function to interface with ConveyLinx Aix Controller for 110
      sFB_MCOConveyLinxAixController120 { ExternalAccessible := 'False'; ExternalVisible := 'False'; ExternalWritable := 'False'; S7_SetPoint := 'False'} : "FB_MCOConveyLinxAixController";   // Function to interface with ConveyLinx Aix Controller for 120
      sFB_MCOConveyLinxAixController121 { ExternalAccessible := 'False'; ExternalVisible := 'False'; ExternalWritable := 'False'; S7_SetPoint := 'False'} : "FB_MCOConveyLinxAixController";   // Function to interface with ConveyLinx Aix Controller for 121
      sFB_MCOConveyLinxAixController210 { ExternalAccessible := 'False'; ExternalVisible := 'False'; ExternalWritable := 'False'; S7_SetPoint := 'False'} : "FB_MCOConveyLinxAixController";   // Function to interface with ConveyLinx Aix Controller for 210
      sFB_MCOConveyLinxAixController220 { ExternalAccessible := 'False'; ExternalVisible := 'False'; ExternalWritable := 'False'; S7_SetPoint := 'False'} : "FB_MCOConveyLinxAixController";   // Function to interface with ConveyLinx Aix Controller for 220
      sFB_MCOConveyLinxAixController221 { ExternalAccessible := 'False'; ExternalVisible := 'False'; ExternalWritable := 'False'; S7_SetPoint := 'False'} : "FB_MCOConveyLinxAixController";   // Function to interface with ConveyLinx Aix Controller for 221
      sFB_MCOConveyLinxAixController230 { ExternalAccessible := 'False'; ExternalVisible := 'False'; ExternalWritable := 'False'; S7_SetPoint := 'False'} : "FB_MCOConveyLinxAixController";   // Function to interface with ConveyLinx Aix Controller for 230
      sFB_MCOConveyLinxAixController240 { ExternalAccessible := 'False'; ExternalVisible := 'False'; ExternalWritable := 'False'; S7_SetPoint := 'False'} : "FB_MCOConveyLinxAixController";   // Function to interface with ConveyLinx Aix Controller for 240
      sFB_MCOConveyLinxAixController250 { ExternalAccessible := 'False'; ExternalVisible := 'False'; ExternalWritable := 'False'; S7_SetPoint := 'False'} : "FB_MCOConveyLinxAixController";   // Function to interface with ConveyLinx Aix Controller for 250
      sFB_MCOConveyLinxAixController260 { ExternalAccessible := 'False'; ExternalVisible := 'False'; ExternalWritable := 'False'; S7_SetPoint := 'False'} : "FB_MCOConveyLinxAixController";   // Function to interface with ConveyLinx Aix Controller for 260
      sFB_MCOConveyLinxAixController270 { ExternalAccessible := 'False'; ExternalVisible := 'False'; ExternalWritable := 'False'; S7_SetPoint := 'False'} : "FB_MCOConveyLinxAixController";   // Function to interface with ConveyLinx Aix Controller for 270
      sFB_MCOConveyLinxAixController280 { ExternalAccessible := 'False'; ExternalVisible := 'False'; ExternalWritable := 'False'; S7_SetPoint := 'False'} : "FB_MCOConveyLinxAixController";   // Function to interface with ConveyLinx Aix Controller for 280
      sFB_MCOConveyLinxAixController290 { ExternalAccessible := 'False'; ExternalVisible := 'False'; ExternalWritable := 'False'; S7_SetPoint := 'False'} : "FB_MCOConveyLinxAixController";   // Function to interface with ConveyLinx Aix Controller for 290
      sFB_MCOConveyLinxAixController291 { ExternalAccessible := 'False'; ExternalVisible := 'False'; ExternalWritable := 'False'; S7_SetPoint := 'False'} : "FB_MCOConveyLinxAixController";   // Function to interface with ConveyLinx Aix Controller for 291
      sFB_MCOConveyLinxAixController300 { ExternalAccessible := 'False'; ExternalVisible := 'False'; ExternalWritable := 'False'; S7_SetPoint := 'False'} : "FB_MCOConveyLinxAixController";   // Function to interface with ConveyLinx Aix Controller for 300
      sFB_MCOConveyLinxAixController410 { ExternalAccessible := 'False'; ExternalVisible := 'False'; ExternalWritable := 'False'; S7_SetPoint := 'False'} : "FB_MCOConveyLinxAixController";   // Function to interface with ConveyLinx Aix Controller for 410
      sFB_MCOConveyLinxAixController420 { ExternalAccessible := 'False'; ExternalVisible := 'False'; ExternalWritable := 'False'; S7_SetPoint := 'False'} : "FB_MCOConveyLinxAixController";   // Function to interface with ConveyLinx Aix Controller for 420
      sFB_MCOConveyLinxAixController421 { ExternalAccessible := 'False'; ExternalVisible := 'False'; ExternalWritable := 'False'; S7_SetPoint := 'False'} : "FB_MCOConveyLinxAixController";   // Function to interface with ConveyLinx Aix Controller for 421
      sFB_MCOConveyLinxAixController430 { ExternalAccessible := 'False'; ExternalVisible := 'False'; ExternalWritable := 'False'; S7_SetPoint := 'False'} : "FB_MCOConveyLinxAixController";   // Function to interface with ConveyLinx Aix Controller for 430
      sFB_MCOConveyLinxAixController440 { ExternalAccessible := 'False'; ExternalVisible := 'False'; ExternalWritable := 'False'; S7_SetPoint := 'False'} : "FB_MCOConveyLinxAixController";   // Function to interface with ConveyLinx Aix Controller for 440
      sFB_MCOConveyLinxAixController450 { ExternalAccessible := 'False'; ExternalVisible := 'False'; ExternalWritable := 'False'; S7_SetPoint := 'False'} : "FB_MCOConveyLinxAixController";   // Function to interface with ConveyLinx Aix Controller for 450
      sFB_MCOConveyLinxAixController460 { ExternalAccessible := 'False'; ExternalVisible := 'False'; ExternalWritable := 'False'; S7_SetPoint := 'False'} : "FB_MCOConveyLinxAixController";   // Function to interface with ConveyLinx Aix Controller for 460
      sFB_MCOConveyLinxAixController470 { ExternalAccessible := 'False'; ExternalVisible := 'False'; ExternalWritable := 'False'; S7_SetPoint := 'False'} : "FB_MCOConveyLinxAixController";   // Function to interface with ConveyLinx Aix Controller for 470
      sFB_MCOConveyLinxAixController480 { ExternalAccessible := 'False'; ExternalVisible := 'False'; ExternalWritable := 'False'; S7_SetPoint := 'False'} : "FB_MCOConveyLinxAixController";   // Function to interface with ConveyLinx Aix Controller for 480
      sFB_MCOConveyLinxAixController490 { ExternalAccessible := 'False'; ExternalVisible := 'False'; ExternalWritable := 'False'; S7_SetPoint := 'False'} : "FB_MCOConveyLinxAixController";   // Function to interface with ConveyLinx Aix Controller for 490
      sFB_MCOConveyLinxAixController491 { ExternalAccessible := 'False'; ExternalVisible := 'False'; ExternalWritable := 'False'; S7_SetPoint := 'False'} : "FB_MCOConveyLinxAixController";   // Function to interface with ConveyLinx Aix Controller for 491
      sFB_MCOConveyLinxAixController500 { ExternalAccessible := 'False'; ExternalVisible := 'False'; ExternalWritable := 'False'; S7_SetPoint := 'False'} : "FB_MCOConveyLinxAixController";   // Function to interface with ConveyLinx Aix Controller for 500
      sFB_MCOConveyLinxAixController610 { ExternalAccessible := 'False'; ExternalVisible := 'False'; ExternalWritable := 'False'; S7_SetPoint := 'False'} : "FB_MCOConveyLinxAixController";   // Function to interface with ConveyLinx Aix Controller for 610
      sFB_MCOConveyLinxAixController611 { ExternalAccessible := 'False'; ExternalVisible := 'False'; ExternalWritable := 'False'; S7_SetPoint := 'False'} : "FB_MCOConveyLinxAixController";   // Function to interface with ConveyLinx Aix Controller for 611
      sFB_MCOConveyLinxAixController620 { ExternalAccessible := 'False'; ExternalVisible := 'False'; ExternalWritable := 'False'; S7_SetPoint := 'False'} : "FB_MCOConveyLinxAixController";   // Function to interface with ConveyLinx Aix Controller for 620
      sFB_MCOConveyLinxAixController630 { ExternalAccessible := 'False'; ExternalVisible := 'False'; ExternalWritable := 'False'; S7_SetPoint := 'False'} : "FB_MCOConveyLinxAixController";   // Function to interface with ConveyLinx Aix Controller for 630
      sFB_MCOConveyLinxAixController640 { ExternalAccessible := 'False'; ExternalVisible := 'False'; ExternalWritable := 'False'; S7_SetPoint := 'False'} : "FB_MCOConveyLinxAixController";   // Function to interface with ConveyLinx Aix Controller for 630
      sFB_RightAngledTransfer121 { ExternalAccessible := 'False'; ExternalVisible := 'False'; ExternalWritable := 'False'; S7_SetPoint := 'False'} : "FB_RightAngledTransfer";   // Funtion to control 121 RAT
      sFB_RightAngledTransfer221 { ExternalAccessible := 'False'; ExternalVisible := 'False'; ExternalWritable := 'False'; S7_SetPoint := 'False'} : "FB_RightAngledTransfer";   // Funtion to control 221 RAT
      sFB_RightAngledTransfer291 { ExternalAccessible := 'False'; ExternalVisible := 'False'; ExternalWritable := 'False'; S7_SetPoint := 'False'} : "FB_RightAngledTransfer";   // Funtion to control 291 RAT
      sFB_RightAngledTransfer421 { ExternalAccessible := 'False'; ExternalVisible := 'False'; ExternalWritable := 'False'; S7_SetPoint := 'False'} : "FB_RightAngledTransfer";   // Funtion to control 421 RAT
      sFB_RightAngledTransfer491 { ExternalAccessible := 'False'; ExternalVisible := 'False'; ExternalWritable := 'False'; S7_SetPoint := 'False'} : "FB_RightAngledTransfer";   // Funtion to control 491 RAT
      sFB_RightAngledTransfer611 { ExternalAccessible := 'False'; ExternalVisible := 'False'; ExternalWritable := 'False'; S7_SetPoint := 'False'} : "FB_RightAngledTransfer";   // Funtion to control 611 RAT
      sFB_CountActiveInputs_Left { ExternalAccessible := 'False'; ExternalVisible := 'False'; ExternalWritable := 'False'; S7_SetPoint := 'False'} : "FB_CountActiveInputs";   // Count free positions on left station
      sFB_CountActiveInputs_Right { ExternalAccessible := 'False'; ExternalVisible := 'False'; ExternalWritable := 'False'; S7_SetPoint := 'False'} : "FB_CountActiveInputs";   // Count free positions on right station
      sFB_CognexDM280 { ExternalAccessible := 'False'; ExternalVisible := 'False'; ExternalWritable := 'False'; S7_SetPoint := 'False'} : "FB_CognexDM260";   // Cognex camera function block conveyor 280
      sFB_CognexDM480 { ExternalAccessible := 'False'; ExternalVisible := 'False'; ExternalWritable := 'False'; S7_SetPoint := 'False'} : "FB_CognexDM260";   // Cognex camera function block conveyor 480
      ss_Barcode280 { ExternalAccessible := 'False'; ExternalVisible := 'False'; ExternalWritable := 'False'} : String;
      ss_Barcode480 { ExternalAccessible := 'False'; ExternalVisible := 'False'; ExternalWritable := 'False'} : String;
      si_DestinationA121 { ExternalAccessible := 'False'; ExternalVisible := 'False'; ExternalWritable := 'False'} : Int;   // Destination for 121 RAT
      si_DestinationA291 { ExternalAccessible := 'False'; ExternalVisible := 'False'; ExternalWritable := 'False'} : Int;   // Destination for 291 RAT
      si_DestinationA491 { ExternalAccessible := 'False'; ExternalVisible := 'False'; ExternalWritable := 'False'} : Int;   // Destination for 491 RAT
      sx_LastFrom120Right { ExternalAccessible := 'False'; ExternalVisible := 'False'; ExternalWritable := 'False'} : Bool;   // Bit indicating that last divert on RAT 121 was to the right
   END_VAR

   VAR_TEMP
      tUDT_dummyHandshake : "UDT_ConveyorHandshake";   // Dummy Handshake structure
      tUDT_DummyBladeStop : "UDT_ValveInterface";
      tw_dummy : Word;
      tx_dummy : Bool;   // Dummy bool
   END_VAR


BEGIN
	(*
	----------------------------------------------------------------------------------------

	Version history:s
	Date        | Version   | Author        | Remark
	----------------------------------------------------------------------------------------
	22/01/2024  | 0.1       | J.Majer       | Block interface and structure created
	23/02/2024  | 0.2       | R. Pieczonka  | Initial version
	26/02/2024  | 0.3       | S. Nieswiec   | Updated to new library blocks, added HardwareOk input
	18/03/2024  | 0.4       | S. Nieswiec   | Adjusting comments and variable names
	29/03/2024  | 0.5       | S.Nieswiec R. Pieczonka | Added MCOs, PEC changes etc.
	08/05/2024  | 0.6       | S.Nieswiec    | New MCO block
	08/05/2024  | 0.7       | K. Pokorski   | Added displacement
	15/05/2024  | 0.8       | S. Nieswiec   | Clean up, adjusting comments etc.
	08/06/2024  | 0.9       | S. Nieswiec   | New MCO, Displacement and RAT blocks, interface update
	14/06/2024  | 0.10      | S. Nieswiec   | Changed direct sensor inputs to statuses
	*)

	REGION 1 - Initial

	    REGION 1.1 - Counters

	        REGION 1.1.1 - Free slots at left station
	            IF #iUDT_Configuration.GlobalConfig.LeftStationExists THEN
	                #sFB_CountActiveInputs_Left(ix_Input1 := FALSE,//#iUDT_MotorInput440.AllSensorPortInputs.LeftSensor,
	                                            ix_Input2 := #iqUDT_WorkstationStatus."450".PEC_EoS.PEC,
	                                            ix_Input3 := #iqUDT_WorkstationStatus."460".PEC_EoS.PEC,
	                                            ix_Input4 := #iqUDT_WorkstationStatus."480".PEC_EoS.PEC,
	                                            ix_Input5 := #iqUDT_WorkstationStatus."421".PEC_EoS.PEC,
	                                            ix_Input6 := #iqUDT_WorkstationStatus."410".PEC_EoS.PEC);
	            END_IF;

	        END_REGION

	        REGION 1.1.2 - Free slots at right station
	            IF #iUDT_Configuration.GlobalConfig.RightStationExists THEN
	                #sFB_CountActiveInputs_Right(ix_Input1 := FALSE, //#iUDT_MotorInput240.AllSensorPortInputs.LeftSensor,
	                                             ix_Input2 := #iqUDT_WorkstationStatus."250".PEC_EoS.PEC,
	                                             ix_Input3 := #iqUDT_WorkstationStatus."260".PEC_EoS.PEC,
	                                             ix_Input4 := #iqUDT_WorkstationStatus."280".PEC_EoS.PEC,
	                                             ix_Input5 := #iqUDT_WorkstationStatus."221".PEC_EoS.PEC,
	                                             ix_Input6 := #iqUDT_WorkstationStatus."210".PEC_EoS.PEC);
	            END_IF;

	        END_REGION
	    END_REGION

	END_REGION

	REGION 2 - Destinations
	    // Reconsider that logic
	    // Destination FOR 121 RAT depending on existing stations, free spots on each side AND last divert destination
	    IF #iUDT_Configuration.GlobalConfig.LeftStationExists AND NOT #iUDT_Configuration.GlobalConfig.RightStationExists THEN

	        #si_DestinationA121 := 2;

	    ELSIF NOT #iUDT_Configuration.GlobalConfig.LeftStationExists AND #iUDT_Configuration.GlobalConfig.RightStationExists THEN

	        #si_DestinationA121 := 1;

	    ELSIF #iUDT_Configuration.GlobalConfig.LeftStationExists AND #iUDT_Configuration.GlobalConfig.RightStationExists THEN

	        IF #sFB_RightAngledTransfer121.qx_ExternalSendRequestC THEN  //check where was last divert
	            #sx_LastFrom120Right := 1;
	        END_IF;
	        IF #sFB_RightAngledTransfer121.qx_ExternalSendRequestD THEN
	            #sx_LastFrom120Right := 0;
	        END_IF;

	        IF #sFB_CountActiveInputs_Left.qi_ActiveInputsCount > #sFB_CountActiveInputs_Right.qi_ActiveInputsCount AND #iqUDT_WorkstationStatus."410".PEC_EoS.PEC
	            OR (#sFB_CountActiveInputs_Left.qi_ActiveInputsCount = #sFB_CountActiveInputs_Right.qi_ActiveInputsCount
	            AND #sx_LastFrom120Right
	            AND #sFB_CountActiveInputs_Left.qi_ActiveInputsCount <> 0
	            AND #iqUDT_WorkstationStatus."410".PEC_EoS.PEC)
	        THEN
	            #si_DestinationA121 := 2;

	        ELSIF #sFB_CountActiveInputs_Right.qi_ActiveInputsCount <> 0
	            AND #iqUDT_WorkstationStatus."210".PEC_EoS.PEC THEN
	            #si_DestinationA121 := 1;
	        ELSE
	            #si_DestinationA121 := 0;
	        END_IF;
	    END_IF;

	    //Destination for 291 RAT divert out of station after Done request
	    IF #ix_Done490 AND NOT #iqUDT_WorkstationStatus."291".PEC_EoS.PEC THEN
	        #si_DestinationA291 := 1;
	    ELSE
	        #si_DestinationA291 := 0;
	    END_IF;

	    //Destination for 491 RAT RAT divert out of station after Done request
	    IF #ix_Done290 AND NOT #iqUDT_WorkstationStatus."491".PEC_EoS.PEC THEN
	        #si_DestinationA491 := 1;
	    ELSE
	        #si_DestinationA491 := 0;
	    END_IF;

	END_REGION

	REGION 3 - Middle line
	    REGION 010

	        REGION Displacement
	            #sFB_Displacement010(#sUDT_Interface010);
	        END_REGION

	        REGION EoS

	            #sFB_PEC010(ix_PEC := #iUDT_MotorInput010.AllSensorPortInputs.LeftSensor,
	                        iUDT_PECConfiguration := #iUDT_Configuration."010".PEC_EoS,
	                        qUDT_HMIStatus => #iqUDT_WorkstationStatus."010".PEC_EoS,
	                        iqUDT_ConveyorInterface := #sUDT_Interface010,
	                        iqUDT_PECStatistics := #iqUDT_WorkstationStatistics."010".PEC_EoS);

	        END_REGION

	        REGION Conveyor

	            #sFB_Conveyor010(iUDT_ConveyorConfiguration := #iUDT_Configuration."010".Conveyor,
	                             idi_PECEoSDistance := #iUDT_Configuration."010".PEC_EoS.Distance,
	                             idi_PECBoSDistance := 0,
	                             ii_ExternalSpeed := 0,
	                             ix_SafetyOk := #ix_SafetyOk,
	                             ix_24vOk := #ix_24vOk,
	                             ix_400vOk := #ix_400vOk,
	                             ix_HardwareOk := #ix_HardwareOk,
	                             ix_PECEoS := #iqUDT_WorkstationStatus."010".PEC_EoS.PEC,
	                             ix_PECBoS := TRUE,
	                             ix_ReverseDirection := FALSE,
	                             ix_ExternalRequestDieBack := FALSE,
	                             ix_ExternalRequestHold := FALSE,
	                             ix_ResetEnergySave := FALSE,
	                             qUDT_HMIStatus => #iqUDT_WorkstationStatus."010".Conveyor,
	                             qUDT_Status => #iqUDT_WorkstationCommonStatus."010",
	                             iqUDT_EquipmentControl := #iqUDT_EquipmentControl,
	                             iqUDT_ConveyorCommand := #iqUDT_WorkstationCommands."010".Conveyor,
	                             iqUDT_ConveyorInterface := #sUDT_Interface010,
	                             iqUDT_HandShakeUp := #iqUDT_HandshakeUpstream010,
	                             iqUDT_HandShake := #sUDT_Handshake010,
	                             iqUDT_Statistics := #iqUDT_WorkstationStatistics."010".Conveyor);

	        END_REGION

	        REGION MCO

	            #sFB_MCOConveyLinxAixController010(iUDT_AixConfig := #iUDT_Configuration."010".MCO_M01,
	                                               iUDT_AixInputsModule := #iUDT_MotorInput010,
	                                               ix_24vOk := #ix_24vOk,
	                                               ix_SimulationModeActive := "DB_Memory".Simulation,
	                                               ii_MotorPositionId := 1,
	                                               qUDT_HMIStatus => #iqUDT_WorkstationStatus."010".MCO_M01,
	                                               iqUDT_AixOutputsModule := #qUDT_MotorOutput010,
	                                               iqUDT_ConveyorInterface := #sUDT_Interface010,
	                                               iqUDT_MCOStatistics := #iqUDT_WorkstationStatistics."010".MCO_M01);
	        END_REGION

	    END_REGION

	    REGION 020

	        REGION Displacement
	            #sFB_Displacement020(#sUDT_Interface020);
	        END_REGION

	        REGION EoS

	            #sFB_PEC020(ix_PEC := #iUDT_MotorInput010.AllSensorPortInputs.RightSensor,
	                        iUDT_PECConfiguration := #iUDT_Configuration."020".PEC_EoS,
	                        qUDT_HMIStatus => #iqUDT_WorkstationStatus."020".PEC_EoS,
	                        iqUDT_ConveyorInterface := #sUDT_Interface020,
	                        iqUDT_PECStatistics := #iqUDT_WorkstationStatistics."020".PEC_EoS);

	        END_REGION
	        REGION Conveyor

	            #sFB_Conveyor020(iUDT_ConveyorConfiguration := #iUDT_Configuration."020".Conveyor,
	                             idi_PECEoSDistance := #iUDT_Configuration."020".PEC_EoS.Distance,
	                             idi_PECBoSDistance := 0,
	                             ii_ExternalSpeed := 0,
	                             ix_SafetyOk := #ix_SafetyOk,
	                             ix_24vOk := #ix_24vOk,
	                             ix_400vOk := #ix_400vOk,
	                             ix_HardwareOk := #ix_HardwareOk,
	                             ix_PECEoS := #iqUDT_WorkstationStatus."020".PEC_EoS.PEC,
	                             ix_PECBoS := TRUE,
	                             ix_ReverseDirection := FALSE,
	                             ix_ExternalRequestDieBack := FALSE,
	                             ix_ExternalRequestHold := FALSE,
	                             ix_ResetEnergySave := FALSE,
	                             qUDT_HMIStatus => #iqUDT_WorkstationStatus."020".Conveyor,
	                             qUDT_Status => #iqUDT_WorkstationCommonStatus."020",
	                             iqUDT_EquipmentControl := #iqUDT_EquipmentControl,
	                             iqUDT_ConveyorCommand := #iqUDT_WorkstationCommands."020".Conveyor,
	                             iqUDT_ConveyorInterface := #sUDT_Interface020,
	                             iqUDT_HandShakeUp := #sUDT_Handshake010,
	                             iqUDT_HandShake := #sUDT_Handshake020,
	                             iqUDT_Statistics := #iqUDT_WorkstationStatistics."020".Conveyor);

	        END_REGION

	        REGION MCO

	            #sFB_MCOConveyLinxAixController020(iUDT_AixConfig := #iUDT_Configuration."020".MCO_M01,
	                                               iUDT_AixInputsModule := #iUDT_MotorInput010,
	                                               ix_24vOk := #ix_24vOk,
	                                               ix_SimulationModeActive := "DB_Memory".Simulation,
	                                               ii_MotorPositionId := 2,
	                                               qUDT_HMIStatus => #iqUDT_WorkstationStatus."020".MCO_M01,
	                                               iqUDT_AixOutputsModule := #qUDT_MotorOutput010,
	                                               iqUDT_ConveyorInterface := #sUDT_Interface020,
	                                               iqUDT_MCOStatistics := #iqUDT_WorkstationStatistics."020".MCO_M01);
	        END_REGION

	    END_REGION

	    REGION 030

	        REGION Displacement
	            #sFB_Displacement030(#sUDT_Interface030);
	        END_REGION

	        REGION Conveyor

	            #sFB_Conveyor030(iUDT_ConveyorConfiguration := #iUDT_Configuration."030".Conveyor,
	                             idi_PECEoSDistance := 0,
	                             idi_PECBoSDistance := 0,
	                             ii_ExternalSpeed := 0,
	                             ix_SafetyOk := #ix_SafetyOk,
	                             ix_24vOk := #ix_24vOk,
	                             ix_400vOk := #ix_400vOk,
	                             ix_HardwareOk := #ix_HardwareOk,
	                             ix_PECEoS := TRUE,
	                             ix_PECBoS := TRUE,
	                             ix_ReverseDirection := FALSE,
	                             ix_ExternalRequestDieBack := FALSE,
	                             ix_ExternalRequestHold := FALSE,
	                             ix_ResetEnergySave := FALSE,
	                             qUDT_HMIStatus => #iqUDT_WorkstationStatus."030".Conveyor,
	                             qUDT_Status => #iqUDT_WorkstationCommonStatus."030",
	                             iqUDT_EquipmentControl := #iqUDT_EquipmentControl,
	                             iqUDT_ConveyorCommand := #iqUDT_WorkstationCommands."030".Conveyor,
	                             iqUDT_ConveyorInterface := #sUDT_Interface030,
	                             iqUDT_HandShakeUp := #sUDT_Handshake020,
	                             iqUDT_HandShake := #sUDT_Handshake030,
	                             iqUDT_Statistics := #iqUDT_WorkstationStatistics."030".Conveyor);

	        END_REGION
	        REGION MCO

	            #sFB_MCOConveyLinxAixController030(iUDT_AixConfig := #iUDT_Configuration."030".MCO_M01,
	                                               iUDT_AixInputsModule := #iUDT_MotorInput030,
	                                               ix_24vOk := #ix_24vOk,
	                                               ix_SimulationModeActive := "DB_Memory".Simulation,
	                                               ii_MotorPositionId := 1,
	                                               qUDT_HMIStatus => #iqUDT_WorkstationStatus."030".MCO_M01,
	                                               iqUDT_AixOutputsModule := #qUDT_MotorOutput030,
	                                               iqUDT_ConveyorInterface := #sUDT_Interface030,
	                                               iqUDT_MCOStatistics := #iqUDT_WorkstationStatistics."030".MCO_M01);
	        END_REGION
	    END_REGION

	    REGION 040

	        REGION Displacement
	            #sFB_Displacement040(#sUDT_Interface040);
	        END_REGION

	        REGION EoS

	            #sFB_PEC040(ix_PEC := #iUDT_MotorInput040.AllSensorPortInputs.LeftSensor,
	                        iUDT_PECConfiguration := #iUDT_Configuration."040".PEC_EoS,
	                        qUDT_HMIStatus => #iqUDT_WorkstationStatus."040".PEC_EoS,
	                        iqUDT_ConveyorInterface := #sUDT_Interface040,
	                        iqUDT_PECStatistics := #iqUDT_WorkstationStatistics."040".PEC_EoS);

	        END_REGION
	        REGION Conveyor

	            #sFB_Conveyor040(iUDT_ConveyorConfiguration := #iUDT_Configuration."040".Conveyor,
	                             idi_PECEoSDistance := #iUDT_Configuration."040".PEC_EoS.Distance,
	                             idi_PECBoSDistance := 0,
	                             ii_ExternalSpeed := 0,
	                             ix_SafetyOk := #ix_SafetyOk,
	                             ix_24vOk := #ix_24vOk,
	                             ix_400vOk := #ix_400vOk,
	                             ix_HardwareOk := #ix_HardwareOk,
	                             ix_PECEoS := #iqUDT_WorkstationStatus."040".PEC_EoS.PEC,
	                             ix_PECBoS := TRUE,
	                             ix_ReverseDirection := FALSE,
	                             ix_ExternalRequestDieBack := FALSE,
	                             ix_ExternalRequestHold := FALSE,
	                             ix_ResetEnergySave := FALSE,
	                             qUDT_HMIStatus => #iqUDT_WorkstationStatus."040".Conveyor,
	                             qUDT_Status => #iqUDT_WorkstationCommonStatus."040",
	                             iqUDT_EquipmentControl := #iqUDT_EquipmentControl,
	                             iqUDT_ConveyorCommand := #iqUDT_WorkstationCommands."040".Conveyor,
	                             iqUDT_ConveyorInterface := #sUDT_Interface040,
	                             iqUDT_HandShakeUp := #sUDT_Handshake030,
	                             iqUDT_HandShake := #sUDT_Handshake040,
	                             iqUDT_Statistics := #iqUDT_WorkstationStatistics."040".Conveyor);

	        END_REGION

	        REGION MCO

	            #sFB_MCOConveyLinxAixController040(iUDT_AixConfig := #iUDT_Configuration."040".MCO_M01,
	                                               iUDT_AixInputsModule := #iUDT_MotorInput040,
	                                               ix_24vOk := #ix_24vOk,
	                                               ix_SimulationModeActive := "DB_Memory".Simulation,
	                                               ii_MotorPositionId := 1,
	                                               qUDT_HMIStatus => #iqUDT_WorkstationStatus."040".MCO_M01,
	                                               iqUDT_AixOutputsModule := #qUDT_MotorOutput040,
	                                               iqUDT_ConveyorInterface := #sUDT_Interface040,
	                                               iqUDT_MCOStatistics := #iqUDT_WorkstationStatistics."040".MCO_M01);
	        END_REGION
	    END_REGION

	    REGION 050

	        REGION Displacement
	            #sFB_Displacement050(#sUDT_Interface050);
	        END_REGION

	        REGION EoS

	            #sFB_PEC050(ix_PEC := #iUDT_MotorInput050.AllSensorPortInputs.LeftSensor,
	                        iUDT_PECConfiguration := #iUDT_Configuration."050".PEC_EoS,
	                        qUDT_HMIStatus => #iqUDT_WorkstationStatus."050".PEC_EoS,
	                        iqUDT_ConveyorInterface := #sUDT_Interface050,
	                        iqUDT_PECStatistics := #iqUDT_WorkstationStatistics."050".PEC_EoS);

	        END_REGION
	        REGION Conveyor

	            #sFB_Conveyor050(iUDT_ConveyorConfiguration := #iUDT_Configuration."050".Conveyor,
	                             idi_PECEoSDistance := #iUDT_Configuration."050".PEC_EoS.Distance,
	                             idi_PECBoSDistance := 0,
	                             ii_ExternalSpeed := 0,
	                             ix_SafetyOk := #ix_SafetyOk,
	                             ix_24vOk := #ix_24vOk,
	                             ix_400vOk := #ix_400vOk,
	                             ix_HardwareOk := #ix_HardwareOk,
	                             ix_PECEoS := #iqUDT_WorkstationStatus."050".PEC_EoS.PEC,
	                             ix_PECBoS := TRUE,
	                             ix_ReverseDirection := FALSE,
	                             ix_ExternalRequestDieBack := FALSE,
	                             ix_ExternalRequestHold := FALSE,
	                             ix_ResetEnergySave := FALSE,
	                             qUDT_HMIStatus => #iqUDT_WorkstationStatus."050".Conveyor,
	                             qUDT_Status => #iqUDT_WorkstationCommonStatus."050",
	                             iqUDT_EquipmentControl := #iqUDT_EquipmentControl,
	                             iqUDT_ConveyorCommand := #iqUDT_WorkstationCommands."050".Conveyor,
	                             iqUDT_ConveyorInterface := #sUDT_Interface050,
	                             iqUDT_HandShakeUp := #sUDT_Handshake040,
	                             iqUDT_HandShake := #sUDT_Handshake050,
	                             iqUDT_Statistics := #iqUDT_WorkstationStatistics."050".Conveyor);

	        END_REGION

	        REGION MCO

	            #sFB_MCOConveyLinxAixController050(iUDT_AixConfig := #iUDT_Configuration."050".MCO_M01,
	                                               iUDT_AixInputsModule := #iUDT_MotorInput050,
	                                               ix_24vOk := #ix_24vOk,
	                                               ix_SimulationModeActive := "DB_Memory".Simulation,
	                                               ii_MotorPositionId := 1,
	                                               qUDT_HMIStatus => #iqUDT_WorkstationStatus."050".MCO_M01,
	                                               iqUDT_AixOutputsModule := #qUDT_MotorOutput050,
	                                               iqUDT_ConveyorInterface := #sUDT_Interface050,
	                                               iqUDT_MCOStatistics := #iqUDT_WorkstationStatistics."050".MCO_M01);
	        END_REGION
	    END_REGION

	    REGION 060

	        REGION Displacement
	            #sFB_Displacement060(#sUDT_Interface060);
	        END_REGION

	        REGION EoS

	            #sFB_PEC060(ix_PEC := #iUDT_MotorInput060.AllSensorPortInputs.LeftSensor,
	                        iUDT_PECConfiguration := #iUDT_Configuration."060".PEC_EoS,
	                        qUDT_HMIStatus => #iqUDT_WorkstationStatus."060".PEC_EoS,
	                        iqUDT_ConveyorInterface := #sUDT_Interface060,
	                        iqUDT_PECStatistics := #iqUDT_WorkstationStatistics."060".PEC_EoS);

	        END_REGION
	        REGION Conveyor

	            #sFB_Conveyor060(iUDT_ConveyorConfiguration := #iUDT_Configuration."060".Conveyor,
	                             idi_PECEoSDistance := #iUDT_Configuration."060".PEC_EoS.Distance,
	                             idi_PECBoSDistance := 0,
	                             ii_ExternalSpeed := 0,
	                             ix_SafetyOk := #ix_SafetyOk,
	                             ix_24vOk := #ix_24vOk,
	                             ix_400vOk := #ix_400vOk,
	                             ix_HardwareOk := #ix_HardwareOk,
	                             ix_PECEoS := #iqUDT_WorkstationStatus."060".PEC_EoS.PEC,
	                             ix_PECBoS := TRUE,
	                             ix_ReverseDirection := FALSE,
	                             ix_ExternalRequestDieBack := FALSE,
	                             ix_ExternalRequestHold := FALSE,
	                             ix_ResetEnergySave := FALSE,
	                             qUDT_HMIStatus => #iqUDT_WorkstationStatus."060".Conveyor,
	                             qUDT_Status => #iqUDT_WorkstationCommonStatus."060",
	                             iqUDT_EquipmentControl := #iqUDT_EquipmentControl,
	                             iqUDT_ConveyorCommand := #iqUDT_WorkstationCommands."060".Conveyor,
	                             iqUDT_ConveyorInterface := #sUDT_Interface060,
	                             iqUDT_HandShakeUp := #sUDT_Handshake050,
	                             iqUDT_HandShake := #sUDT_Handshake060,
	                             iqUDT_Statistics := #iqUDT_WorkstationStatistics."060".Conveyor);

	        END_REGION

	        REGION MCO

	            #sFB_MCOConveyLinxAixController060(iUDT_AixConfig := #iUDT_Configuration."060".MCO_M01,
	                                               iUDT_AixInputsModule := #iUDT_MotorInput060,
	                                               ix_24vOk := #ix_24vOk,
	                                               ix_SimulationModeActive := "DB_Memory".Simulation,
	                                               ii_MotorPositionId := 1,
	                                               qUDT_HMIStatus => #iqUDT_WorkstationStatus."060".MCO_M01,
	                                               iqUDT_AixOutputsModule := #qUDT_MotorOutput060,
	                                               iqUDT_ConveyorInterface := #sUDT_Interface060,
	                                               iqUDT_MCOStatistics := #iqUDT_WorkstationStatistics."060".MCO_M01);
	        END_REGION
	    END_REGION

	    REGION 070

	        REGION Displacement
	            #sFB_Displacement070(#sUDT_Interface070);
	        END_REGION

	        REGION EoS

	            #sFB_PEC070(ix_PEC := #iUDT_MotorInput070.AllSensorPortInputs.LeftSensor,
	                        iUDT_PECConfiguration := #iUDT_Configuration."070".PEC_EoS,
	                        qUDT_HMIStatus => #iqUDT_WorkstationStatus."070".PEC_EoS,
	                        iqUDT_ConveyorInterface := #sUDT_Interface070,
	                        iqUDT_PECStatistics := #iqUDT_WorkstationStatistics."070".PEC_EoS);

	        END_REGION
	        REGION Conveyor

	            #sFB_Conveyor070(iUDT_ConveyorConfiguration := #iUDT_Configuration."070".Conveyor,
	                             idi_PECEoSDistance := #iUDT_Configuration."070".PEC_EoS.Distance,
	                             idi_PECBoSDistance := 0,
	                             ii_ExternalSpeed := 0,
	                             ix_SafetyOk := #ix_SafetyOk,
	                             ix_24vOk := #ix_24vOk,
	                             ix_400vOk := #ix_400vOk,
	                             ix_HardwareOk := #ix_HardwareOk,
	                             ix_PECEoS := #iqUDT_WorkstationStatus."070".PEC_EoS.PEC,
	                             ix_PECBoS := TRUE,
	                             ix_ReverseDirection := FALSE,
	                             ix_ExternalRequestDieBack := FALSE,
	                             ix_ExternalRequestHold := FALSE,
	                             ix_ResetEnergySave := FALSE,
	                             qUDT_HMIStatus => #iqUDT_WorkstationStatus."070".Conveyor,
	                             qUDT_Status => #iqUDT_WorkstationCommonStatus."070",
	                             iqUDT_EquipmentControl := #iqUDT_EquipmentControl,
	                             iqUDT_ConveyorCommand := #iqUDT_WorkstationCommands."070".Conveyor,
	                             iqUDT_ConveyorInterface := #sUDT_Interface070,
	                             iqUDT_HandShakeUp := #sUDT_Handshake060,
	                             iqUDT_HandShake := #sUDT_Handshake070,
	                             iqUDT_Statistics := #iqUDT_WorkstationStatistics."070".Conveyor);

	        END_REGION

	        REGION MCO

	            #sFB_MCOConveyLinxAixController070(iUDT_AixConfig := #iUDT_Configuration."070".MCO_M01,
	                                               iUDT_AixInputsModule := #iUDT_MotorInput070,
	                                               ix_24vOk := #ix_24vOk,
	                                               ix_SimulationModeActive := "DB_Memory".Simulation,
	                                               ii_MotorPositionId := 1,
	                                               qUDT_HMIStatus => #iqUDT_WorkstationStatus."070".MCO_M01,
	                                               iqUDT_AixOutputsModule := #qUDT_MotorOutput070,
	                                               iqUDT_ConveyorInterface := #sUDT_Interface070,
	                                               iqUDT_MCOStatistics := #iqUDT_WorkstationStatistics."070".MCO_M01);
	        END_REGION
	    END_REGION

	    REGION 080

	        REGION Displacement
	            #sFB_Displacement080(#sUDT_Interface080);
	        END_REGION

	        REGION EoS

	            #sFB_PEC080(ix_PEC := #iUDT_MotorInput080.AllSensorPortInputs.LeftSensor,
	                        iUDT_PECConfiguration := #iUDT_Configuration."080".PEC_EoS,
	                        qUDT_HMIStatus => #iqUDT_WorkstationStatus."080".PEC_EoS,
	                        iqUDT_ConveyorInterface := #sUDT_Interface080,
	                        iqUDT_PECStatistics := #iqUDT_WorkstationStatistics."080".PEC_EoS);

	        END_REGION
	        REGION Conveyor

	            #sFB_Conveyor080(iUDT_ConveyorConfiguration := #iUDT_Configuration."080".Conveyor,
	                             idi_PECEoSDistance := #iUDT_Configuration."080".PEC_EoS.Distance,
	                             idi_PECBoSDistance := 0,
	                             ii_ExternalSpeed := 0,
	                             ix_SafetyOk := #ix_SafetyOk,
	                             ix_24vOk := #ix_24vOk,
	                             ix_400vOk := #ix_400vOk,
	                             ix_HardwareOk := #ix_HardwareOk,
	                             ix_PECEoS := #iqUDT_WorkstationStatus."080".PEC_EoS.PEC,
	                             ix_PECBoS := TRUE,
	                             ix_ReverseDirection := FALSE,
	                             ix_ExternalRequestDieBack := FALSE,
	                             ix_ExternalRequestHold := FALSE,
	                             ix_ResetEnergySave := FALSE,
	                             qUDT_HMIStatus => #iqUDT_WorkstationStatus."080".Conveyor,
	                             qUDT_Status => #iqUDT_WorkstationCommonStatus."080",
	                             iqUDT_EquipmentControl := #iqUDT_EquipmentControl,
	                             iqUDT_ConveyorCommand := #iqUDT_WorkstationCommands."080".Conveyor,
	                             iqUDT_ConveyorInterface := #sUDT_Interface080,
	                             iqUDT_HandShakeUp := #sUDT_Handshake070,
	                             iqUDT_HandShake := #sUDT_Handshake080,
	                             iqUDT_Statistics := #iqUDT_WorkstationStatistics."080".Conveyor);

	        END_REGION

	        REGION MCO

	            #sFB_MCOConveyLinxAixController080(iUDT_AixConfig := #iUDT_Configuration."080".MCO_M01,
	                                               iUDT_AixInputsModule := #iUDT_MotorInput080,
	                                               ix_24vOk := #ix_24vOk,
	                                               ix_SimulationModeActive := "DB_Memory".Simulation,
	                                               ii_MotorPositionId := 1,
	                                               qUDT_HMIStatus => #iqUDT_WorkstationStatus."080".MCO_M01,
	                                               iqUDT_AixOutputsModule := #qUDT_MotorOutput080,
	                                               iqUDT_ConveyorInterface := #sUDT_Interface080,
	                                               iqUDT_MCOStatistics := #iqUDT_WorkstationStatistics."080".MCO_M01);
	        END_REGION
	    END_REGION

	    REGION 090

	        REGION Displacement
	            #sFB_Displacement090(#sUDT_Interface090);
	        END_REGION

	        REGION Conveyor

	            #sFB_Conveyor090(iUDT_ConveyorConfiguration := #iUDT_Configuration."090".Conveyor,
	                             idi_PECEoSDistance := 0,
	                             idi_PECBoSDistance := 0,
	                             ii_ExternalSpeed := 0,
	                             ix_SafetyOk := #ix_SafetyOk,
	                             ix_24vOk := #ix_24vOk,
	                             ix_400vOk := #ix_400vOk,
	                             ix_HardwareOk := #ix_HardwareOk,
	                             ix_PECEoS := TRUE,
	                             ix_PECBoS := TRUE,
	                             ix_ReverseDirection := FALSE,
	                             ix_ExternalRequestDieBack := FALSE,
	                             ix_ExternalRequestHold := FALSE,
	                             ix_ResetEnergySave := FALSE,
	                             qUDT_HMIStatus => #iqUDT_WorkstationStatus."090".Conveyor,
	                             qUDT_Status => #iqUDT_WorkstationCommonStatus."090",
	                             iqUDT_EquipmentControl := #iqUDT_EquipmentControl,
	                             iqUDT_ConveyorCommand := #iqUDT_WorkstationCommands."090".Conveyor,
	                             iqUDT_ConveyorInterface := #sUDT_Interface090,
	                             iqUDT_HandShakeUp := #sUDT_Handshake080,
	                             iqUDT_HandShake := #sUDT_Handshake090,
	                             iqUDT_Statistics := #iqUDT_WorkstationStatistics."090".Conveyor);

	        END_REGION
	        REGION MCO

	            #sFB_MCOConveyLinxAixController090(iUDT_AixConfig := #iUDT_Configuration."090".MCO_M01,
	                                               iUDT_AixInputsModule := #iUDT_MotorInput090,
	                                               ix_24vOk := #ix_24vOk,
	                                               ix_SimulationModeActive := "DB_Memory".Simulation,
	                                               ii_MotorPositionId := 1,
	                                               qUDT_HMIStatus => #iqUDT_WorkstationStatus."090".MCO_M01,
	                                               iqUDT_AixOutputsModule := #qUDT_MotorOutput090,
	                                               iqUDT_ConveyorInterface := #sUDT_Interface090,
	                                               iqUDT_MCOStatistics := #iqUDT_WorkstationStatistics."090".MCO_M01);
	        END_REGION
	    END_REGION

	    REGION 100

	        REGION Displacement
	            #sFB_Displacement100(#sUDT_Interface100);
	        END_REGION

	        REGION EoS

	            #sFB_PEC100(ix_PEC := #iUDT_MotorInput100.AllSensorPortInputs.LeftSensor,
	                        iUDT_PECConfiguration := #iUDT_Configuration."100".PEC_EoS,
	                        qUDT_HMIStatus => #iqUDT_WorkstationStatus."100".PEC_EoS,
	                        iqUDT_ConveyorInterface := #sUDT_Interface100,
	                        iqUDT_PECStatistics := #iqUDT_WorkstationStatistics."100".PEC_EoS);

	        END_REGION
	        REGION Conveyor

	            #sFB_Conveyor100(iUDT_ConveyorConfiguration := #iUDT_Configuration."100".Conveyor,
	                             idi_PECEoSDistance := #iUDT_Configuration."100".PEC_EoS.Distance,
	                             idi_PECBoSDistance := 0,
	                             ii_ExternalSpeed := 0,
	                             ix_SafetyOk := #ix_SafetyOk,
	                             ix_24vOk := #ix_24vOk,
	                             ix_400vOk := #ix_400vOk,
	                             ix_HardwareOk := #ix_HardwareOk,
	                             ix_PECEoS := #iqUDT_WorkstationStatus."100".PEC_EoS.PEC,
	                             ix_PECBoS := TRUE,
	                             ix_ReverseDirection := FALSE,
	                             ix_ExternalRequestDieBack := FALSE,
	                             ix_ExternalRequestHold := FALSE,
	                             ix_ResetEnergySave := FALSE,
	                             qUDT_HMIStatus => #iqUDT_WorkstationStatus."100".Conveyor,
	                             qUDT_Status => #iqUDT_WorkstationCommonStatus."100",
	                             iqUDT_EquipmentControl := #iqUDT_EquipmentControl,
	                             iqUDT_ConveyorCommand := #iqUDT_WorkstationCommands."100".Conveyor,
	                             iqUDT_ConveyorInterface := #sUDT_Interface100,
	                             iqUDT_HandShakeUp := #sUDT_Handshake090,
	                             iqUDT_HandShake := #sUDT_Handshake100,
	                             iqUDT_Statistics := #iqUDT_WorkstationStatistics."100".Conveyor);

	        END_REGION

	        REGION MCO

	            #sFB_MCOConveyLinxAixController100(iUDT_AixConfig := #iUDT_Configuration."100".MCO_M01,
	                                               iUDT_AixInputsModule := #iUDT_MotorInput100,
	                                               ix_24vOk := #ix_24vOk,
	                                               ix_SimulationModeActive := "DB_Memory".Simulation,
	                                               ii_MotorPositionId := 1,
	                                               qUDT_HMIStatus => #iqUDT_WorkstationStatus."100".MCO_M01,
	                                               iqUDT_AixOutputsModule := #qUDT_MotorOutput100,
	                                               iqUDT_ConveyorInterface := #sUDT_Interface100,
	                                               iqUDT_MCOStatistics := #iqUDT_WorkstationStatistics."100".MCO_M01);
	        END_REGION
	    END_REGION

	    REGION 110

	        REGION Displacement
	            #sFB_Displacement110(#sUDT_Interface110);
	        END_REGION

	        REGION EoS

	            #sFB_PEC110(ix_PEC := #iUDT_MotorInput110.AllSensorPortInputs.LeftSensor,
	                        iUDT_PECConfiguration := #iUDT_Configuration."110".PEC_EoS,
	                        qUDT_HMIStatus => #iqUDT_WorkstationStatus."110".PEC_EoS,
	                        iqUDT_ConveyorInterface := #sUDT_Interface110,
	                        iqUDT_PECStatistics := #iqUDT_WorkstationStatistics."110".PEC_EoS);

	        END_REGION
	        REGION Conveyor

	            #sUDT_Handshake110.RTR := #sUDT_Handshake110.RTR OR #iqUDT_WorkstationStatus."110".PEC_EoS.PEC;

	            #sFB_Conveyor110(iUDT_ConveyorConfiguration := #iUDT_Configuration."110".Conveyor,
	                             idi_PECEoSDistance := #iUDT_Configuration."110".PEC_EoS.Distance,
	                             idi_PECBoSDistance := 0,
	                             ii_ExternalSpeed := 0,
	                             ix_SafetyOk := #ix_SafetyOk,
	                             ix_24vOk := #ix_24vOk,
	                             ix_400vOk := #ix_400vOk,
	                             ix_HardwareOk := #ix_HardwareOk,
	                             ix_PECEoS := #iqUDT_WorkstationStatus."110".PEC_EoS.PEC,
	                             ix_PECBoS := TRUE,
	                             ix_ReverseDirection := FALSE,
	                             ix_ExternalRequestDieBack := FALSE,
	                             ix_ExternalRequestHold := FALSE,
	                             ix_ResetEnergySave := FALSE,
	                             qUDT_HMIStatus => #iqUDT_WorkstationStatus."110".Conveyor,
	                             qUDT_Status => #iqUDT_WorkstationCommonStatus."110",
	                             iqUDT_EquipmentControl := #iqUDT_EquipmentControl,
	                             iqUDT_ConveyorCommand := #iqUDT_WorkstationCommands."110".Conveyor,
	                             iqUDT_ConveyorInterface := #sUDT_Interface110,
	                             iqUDT_HandShakeUp := #sUDT_Handshake100,
	                             iqUDT_HandShake := #sUDT_Handshake110,
	                             iqUDT_Statistics := #iqUDT_WorkstationStatistics."110".Conveyor);

	        END_REGION
	        REGION MCO

	            #sFB_MCOConveyLinxAixController110(iUDT_AixConfig := #iUDT_Configuration."110".MCO_M01,
	                                               iUDT_AixInputsModule := #iUDT_MotorInput110,
	                                               ix_24vOk := #ix_24vOk,
	                                               ix_SimulationModeActive := "DB_Memory".Simulation,
	                                               ii_MotorPositionId := 1,
	                                               qUDT_HMIStatus => #iqUDT_WorkstationStatus."110".MCO_M01,
	                                               iqUDT_AixOutputsModule := #qUDT_MotorOutput110,
	                                               iqUDT_ConveyorInterface := #sUDT_Interface110,
	                                               iqUDT_MCOStatistics := #iqUDT_WorkstationStatistics."110".MCO_M01);
	        END_REGION
	    END_REGION

	    REGION 120

	        REGION Displacement
	            #sFB_Displacement120(#sUDT_Interface120);
	        END_REGION

	        REGION MCO

	            #sFB_MCOConveyLinxAixController120(iUDT_AixConfig := #iUDT_Configuration."120".MCO_M01,
	                                               iUDT_AixInputsModule := #iUDT_MotorInput120,
	                                               ii_PositionSetpoint := #iqUDT_RATPositioning120.Lower.EndPosition,
	                                               ix_24vOk := #ix_24vOk,
	                                               ix_SimulationModeActive := "DB_Memory".Simulation,
	                                               ii_MotorPositionId := 1,
	                                               ix_StartPositioning := #iqUDT_RATPositioning120.Lower.Start,
	                                               ix_ResetPosition := #iqUDT_RATPositioning120.Lower.ResetPosition,
	                                               qUDT_HMIStatus => #iqUDT_WorkstationStatus."120".MCO_M01,
	                                               qx_Positioned => #iqUDT_RATPositioning120.Lower.Done,
	                                               iqUDT_AixOutputsModule := #qUDT_MotorOutput120,
	                                               iqUDT_ConveyorInterface := #sUDT_Interface120,
	                                               iqUDT_MCOStatistics := #iqUDT_WorkstationStatistics."120".MCO_M01);
	        END_REGION
	    END_REGION

	    REGION 121

	        REGION Displacement
	            #sFB_Displacement121(#sUDT_Interface121);
	        END_REGION

	        REGION RAT

	            #sFB_RightAngledTransfer121(iUDT_Configuration := #iUDT_Configuration."121".RightAngledTransfer,
	                                        iUDT_LowerConveyorConfiguration := #iUDT_Configuration."120".Conveyor,
	                                        iUDT_UpperConveyorConfiguration := #iUDT_Configuration."121".Conveyor,
	                                        iUDT_PECConfiguration := #iUDT_Configuration."120".PEC_EoS,
	                                        ii_DestinationA := #si_DestinationA121,
	                                        ii_DestinationB := 0,
	                                        ii_DestinationC := 0,
	                                        ii_DestinationD := 0,
	                                        ix_HardwareOk := #ix_HardwareOk,
	                                        ix_400vOk := #ix_400vOk,
	                                        ix_24vOk := #ix_24vOk,
	                                        ix_SafetyOk := #ix_SafetyOk,
	                                        ix_AirPressureOk := #ix_AirPressureOk,
	                                        ix_SectionIsDown := #ix_SectionIsDown121,
	                                        ix_SectionIsUp := #ix_SectionIsUp121,
	                                        ix_ConveyorAAuto := #iqUDT_WorkstationCommonStatus."110".AutoON,
	                                        ix_ConveyorBAuto := false,
	                                        ix_ConveyorCAuto := #iqUDT_WorkstationCommonStatus."210".AutoON,
	                                        ix_ConveyorDAuto := #iqUDT_WorkstationCommonStatus."410".AutoON,
	                                        ix_PEC := #iUDT_MotorInput120.AllSensorPortInputs.LeftSensor,
	                                        ix_ExternalReceiveRequestA := NOT #iqUDT_WorkstationStatus."110".PEC_EoS.PEC,
	                                        ix_ExternalReceiveRequestB := FALSE,
	                                        ix_ExternalReceiveRequestC := FALSE,
	                                        ix_ExternalReceiveRequestD := FALSE,
	                                        ix_PECInfeedA := #iqUDT_WorkstationStatus."110".PEC_EoS.PEC,
	                                        ix_PECInfeedB := false,
	                                        ix_PECInfeedC := false,
	                                        ix_PECInfeedD := false,
	                                        qUDT_HMIRATStatus => #iqUDT_WorkstationStatus."121".RightAngledTransfer,
	                                        qUDT_HMIConveyorStatus => #iqUDT_WorkstationStatus."120".Conveyor,
	                                        qUDT_HMIPECStatus => #iqUDT_WorkstationStatus."121".PEC_EoS,
	                                        qUDT_RATStatus => #iqUDT_WorkstationCommonStatus."121",
	                                        qUDT_ConveyorStatus => #iqUDT_WorkstationCommonStatus."120",
	                                        qx_PopupControl => #qx_PopupControl121,
	                                        qx_ExternalSendRequestA => #tx_dummy,
	                                        qx_ExternalSendRequestB => #tx_dummy,
	                                        qx_ExternalSendRequestC => #tx_dummy,
	                                        qx_ExternalSendRequestD => #tx_dummy,
	                                        iqUDT_EquipmentControl := #iqUDT_EquipmentControl,
	                                        iqUDT_RATCommand := #iqUDT_WorkstationCommands."121".RightAngledTransfer,
	                                        iqUDT_ConveyorCommand := #iqUDT_WorkstationCommands."120".Conveyor,
	                                        iqUDT_RATStatistics := #iqUDT_WorkstationStatistics."121".RightAngledTransfer,
	                                        iqUDT_ConveyorStatistics := #iqUDT_WorkstationStatistics."120".Conveyor,
	                                        iqUDT_PECStatistics := #iqUDT_WorkstationStatistics."121".PEC_EoS,
	                                        iqUDT_HandShakeConveyorA := #sUDT_Handshake110,
	                                        iqUDT_HandShakeConveyorB := #tUDT_dummyHandshake,
	                                        iqUDT_HandShakeConveyorC := #sUDT_HandshakeUp121,
	                                        iqUDT_HandShakeConveyorD := #sUDT_Handshake121,
	                                        iqUDT_LowerConveyorInterface := #sUDT_Interface120,
	                                        iqUDT_UpperConveyorInterface := #sUDT_Interface121,
	                                        iqUDT_RATPositioning := #iqUDT_RATPositioning120,
	                                        iqUDT_BladeStopEoSInterface := #tUDT_DummyBladeStop,
	                                        iqUDT_BladeStopBoSInterface := #tUDT_DummyBladeStop);

	        END_REGION

	        REGION MCO

	            #sFB_MCOConveyLinxAixController121(iUDT_AixConfig := #iUDT_Configuration."121".MCO_M01,
	                                               iUDT_AixInputsModule := #iUDT_MotorInput120,
	                                               ix_24vOk := #ix_24vOk,
	                                               ix_SimulationModeActive := "DB_Memory".Simulation,
	                                               ii_MotorPositionId := 2,
	                                               qUDT_HMIStatus => #iqUDT_WorkstationStatus."121".MCO_M01,
	                                               iqUDT_AixOutputsModule := #qUDT_MotorOutput120,
	                                               iqUDT_ConveyorInterface := #sUDT_Interface121,
	                                               iqUDT_MCOStatistics := #iqUDT_WorkstationStatistics."121".MCO_M01);
	        END_REGION

	    END_REGION
	END_REGION

	REGION 4 - Right Station
	    IF #iUDT_Configuration.GlobalConfig.RightStationExists THEN
	        REGION 210

	            REGION Displacement
	                #sFB_Displacement210(#sUDT_Interface210);
	            END_REGION

	            REGION EoS

	                #sFB_PEC210(ix_PEC := #iUDT_MotorInput210.AllSensorPortInputs.LeftSensor,
	                            iUDT_PECConfiguration := #iUDT_Configuration."210".PEC_EoS,
	                            qUDT_HMIStatus => #iqUDT_WorkstationStatus."210".PEC_EoS,
	                            iqUDT_ConveyorInterface := #sUDT_Interface210,
	                            iqUDT_PECStatistics := #iqUDT_WorkstationStatistics."210".PEC_EoS);

	            END_REGION
	            REGION Conveyor

	                #sUDT_Handshake210.RTR := #sUDT_Handshake210.RTR OR #iqUDT_WorkstationStatus."210".PEC_EoS.PEC;

	                #sFB_Conveyor210(iUDT_ConveyorConfiguration := #iUDT_Configuration."210".Conveyor,
	                                 idi_PECEoSDistance := #iUDT_Configuration."210".PEC_EoS.Distance,
	                                 idi_PECBoSDistance := 0,
	                                 ii_ExternalSpeed := 0,
	                                 ix_SafetyOk := #ix_SafetyOk,
	                                 ix_24vOk := #ix_24vOk,
	                                 ix_400vOk := #ix_400vOk,
	                                 ix_HardwareOk := #ix_HardwareOk,
	                                 ix_PECEoS := #iqUDT_WorkstationStatus."210".PEC_EoS.PEC,
	                                 ix_PECBoS := TRUE,
	                                 ix_ReverseDirection := FALSE,
	                                 ix_ExternalRequestDieBack := FALSE,
	                                 ix_ExternalRequestHold := FALSE,
	                                 ix_ResetEnergySave := FALSE,
	                                 qUDT_HMIStatus => #iqUDT_WorkstationStatus."210".Conveyor,
	                                 qUDT_Status => #iqUDT_WorkstationCommonStatus."210",
	                                 iqUDT_EquipmentControl := #iqUDT_EquipmentControl,
	                                 iqUDT_ConveyorCommand := #iqUDT_WorkstationCommands."210".Conveyor,
	                                 iqUDT_ConveyorInterface := #sUDT_Interface210,
	                                 iqUDT_HandShakeUp := #sUDT_HandshakeUp121,
	                                 iqUDT_HandShake := #sUDT_Handshake210,
	                                 iqUDT_Statistics := #iqUDT_WorkstationStatistics."210".Conveyor);

	            END_REGION
	            REGION MCO

